(* CoDeSys 2.3 library: TcBACnetRev12.lib *)
(* Libraries: standard.lib 5.6.98 11:03:02, TcBase.lib 14.5.09 11:14:08, TcSystem.lib 21.1.15 09:22:54, TcUtilities.lib 6.1.15 15:45:04, TcTestAndSet.lib 23.2.09 11:50:08 *)

(* Global variable list: BACnet_Globals *)
VAR_GLOBAL
(* ADS read/write buffer for dynamic sized properties *)
	stBACnet_AdsBuffer		: ST_BACnet_GlobalAdsBuffer; (* 8kByte common ADS buffer used by function blocks that access BACnet over ADS *)
(* global linkable BACnet adapter *)
	fbBACnet_Adapter		: FB_BACnet_Adapter;
(* global visible BACnet adapter reference *)
	pBACnet_Adapter			: POINTER TO FB_BACnet_Adapter;
END_VAR
VAR_GLOBAL CONSTANT
(*********************************************
	Data field maximum
**********************************************)
	BACnet_MaxDayEntry			: UINT := 19;
	BACnet_MaxExSchEntries		: UINT := 9;
	BACnet_MaxTimeValues		: UINT := 9;
	BACnet_MaxObjIdList			: UINT := 1999;
	BACnet_MaxLogBufferEntries	: UINT := 499;
	BACnet_MaxDestinationArray	: UINT := 19;

(*********************************************
	error codes
**********************************************)
	BACnet_ERR_NO_ERROR				: UINT := 0;
	BACnet_ERR_NO_VALID_NET_ID		: UINT := 1;
	BACnet_ERR_WRONG_MAPPING		: UINT := 2;
	BACnet_ERR_OPERATIONAL			: UINT := 3;
	BACnet_ERR_NO_ETH_LINK			: UINT := 4;
	BACnet_ERR_NO_GATEWAY			: UINT := 5;
	BACnet_ERR_WOC_TRIGGER_UNSUP	: UINT := 6;
	BACnet_ERR_WOC_DISABLED			: UINT := 7;
	BACnet_ERR_INVALID_OBJECTID		: UINT := 8;
	BACnet_ERR_INVALID_OBJECTTYPE	: UINT := 10;
	BACnet_ERR_INVALID_CYCLETIME	: UINT := 11;
	BACnet_ERR_INVALID_PARAMETER	: UINT := 12;

(* errors with reset 20.. *)
	BACnet_ERR_PERSISTENT_WRITE		: UINT := 20;
	BACnet_ERR_INVALID_ADS_CONN		: UINT := 21;
	BACnet_ERR_CLIENT_TIMEOUT		: UINT := 22;
	BACnet_ERR_CLIENT_SERVICE		: UINT := 23;
	BACnet_ERR_WOC_TRIGGER_ACTIVE	: UINT := 24;
	BACnet_ERR_REVISION_READ		: UINT := 25;
	BACnet_ERR_PERSISTENT_PLC_WRITE	: UINT := 26;

(* ADS connection errors 30.. *)
	BACnet_ERR_ADS_NO_VALID_NET_ID	: UINT := 30; (* missing a valid Net ID *)
	BACnet_ERR_ADS_Data				: UINT := 31; (* ADS data length is wrong *)
	BACnet_ERR_ADS_Read				: UINT := 32; (* ADS read function was aborted *)
	BACnet_ERR_ADS_Write			: UINT := 33; (* ADS write function was aborted *)
	BACnet_ERR_ADS_ObjType			: UINT := 34; (* object type is wrong *)
	BACnet_ERR_ADS_ObjListEmpty		: UINT := 35; (* object list is empty *)
	BACnet_ERR_ADS_DeviceOP			: UINT := 36; (* device is not operational *)
	BACnet_ERR_ADS_NoDevice			: UINT := 37; (* no device object in object info list *)
	BACnet_ERR_ADS_ObjInstance		: UINT := 38; (* object list info is wrong *)
	BACnet_ERR_ADS_AmsPort			: UINT := 39; (* read AMS port is invalid (<1000) *)
	BACnet_ERR_ADS_ObjectId			: UINT := 40; (* object list info is wrong *)
	BACnet_ERR_ADS_LegacyStack		: UINT := 41; (* revision 6 stack detected (service is available from/above revision 9) *)
	BACnet_ERR_ADS_ObjIdMissmatch	: UINT := 42; (* object ID mapped and object list info are different *)
	BACnet_ERR_ADS_BufferSize		: UINT := 43; (* Property data larger than ADS buffer *)
	BACnet_ERR_ADS_SchedData		: UINT := 44; (* Wrong schedule property data *)
	BACnet_ERR_UnknownEventChoice	: UINT := 45; (* Unknown event choice type *)
	BACnet_ERR_UnknownEntryChoice	: UINT := 46; (* Unknown entry choice type *)
	BACnet_ERR_ADS_TooManyObjects	: UINT := 47; (* List of objects are longer than output list size *)
	BACnet_ERR_ADS_WrongEntrySize	: UINT := 48; (* expected entry size dosn't match read size *)
	BACnet_ERR_ADS_RecipientData	: UINT := 49; (* Invalid recipient data, device type expected *)
	BACnet_ERR_ADS_TooManyEntries	: UINT := 50; (* More entries than expected *)
	BACnet_ERR_ADS_NotEnoughEntries	: UINT := 51; (* Property incomplete, missing entries *)
	BACnet_ERR_ADS_Encoding			: UINT := 52; (* String encoding not supported *)
	BACnet_ERR_ADS_NoServerClient	: UINT := 53; (* Given ADS connection is not an server or client connection (expected bClient or bServer) *)
	BACnet_ERR_ADS_NoNotificationSink: UINT := 54; (* Given ADS connection is not an notification sink connection (expected bNSink) *)

(*********************************************
	other definitions
**********************************************)
	BACnet_ADSTimeOut			: TIME := t#15s;
	BACnet_PlcPersisTimeOut		: TIME := t#2m;
	BACnet_STRING_MAXLENGTH     : INT := 256;
	BACnet_ADSBufferSize		: INT := 8191; (* default 8kByte buffer *)

(* ADS index and groups *)
	BACnet_ADSIGRP_GET_OBJECT_LIST						: UDINT := 16#82400000;
	BACnet_ADSIGRP_CLIENT_COM_PARAMETER					: UDINT := 16#84000000;
	BACnet_ADSIGRP_DEV_R_GETADSPORTBYDEVID				: UDINT := 16#80000047; (* Get AMS Port BY Device ID *)
	BACnet_ADSIGRP_NTFSINK_EVENTNTF_CNT					: UDINT := 16#00000001;
	BACnet_ADSIGRP_NTFSINK_COVNTF_CNT					: UDINT := 16#00000002;
	BACnet_ADSIGRP_NTFSINK_EVENTNTF_READ				: UDINT := 16#00000003;
	BACnet_ADSIGRP_NTFSINK_COVNTF_READ					: UDINT := 16#00000004;
	BACnet_ADSIGRP_NTFSINK_EVENTNTF_DELETE				: UDINT := 16#00000005;
	BACnet_ADSIGRP_NTFSINK_COVNTF_DELETE				: UDINT := 16#00000006;
	BACnet_ADSIGRP_NTFSINK_EVENTNTF_INFO				: UDINT := 16#00000007;
	BACnet_ADSIGRP_NTFSINK_COVNTF_INFO					: UDINT := 16#00000008;
	BACnet_ADSIGRP_WRITE_NTFSINK_EVENTNTF_ACK			: UDINT := 16#00000009;
	BACnet_ADSIGRP_NTFSINK_W_EVENTNTF_ACK_BY_SEQUENCE	: UDINT := 16#0000000A;
	BACnet_ADSIGRP_NTFSINK_W_EVENTNTF_ACK_BY_PARAMETER	: UDINT := 16#0000000B;
	BACnet_ADSIGRP_NTFSINK_R_EVENTNTF_READ_BY_SEQUENCE	: UDINT := 16#0000000C;
	BACnet_ADSIGRP_NTFSINK_R_COVNTF_READ_BY_SEQUENCE	: UDINT := 16#0000000D;
	BACnet_ADSIGRP_NTFSINK_R_EVENTNTF_DELETE_BY_SEQUENCE: UDINT := 16#0000000E;
	BACnet_ADSIGRP_NTFSINK_R_COVNTF_DELETE_BY_SEQUENCE	: UDINT := 16#0000000F;


(* Object specifications *)
	arrBACnet_ObjectTypeNameShort : ARRAY[0..BACnetObjectType_ZCount] OF STRING(5) :=
		'AI' (* BACnetObjectType_AnalogInput :=0 *),
		'AO' (* BACnetObjectType_AnalogOutput :=1 *),
		'AV' (* BACnetObjectType_AnalogValue :=2 *),
		'BI' (* BACnetObjectType_BinaryInput :=3 *),
		'BO' (* BACnetObjectType_BinaryOutput :=4 *),
		'BV' (* BACnetObjectType_BinaryValue :=5 *),
		'CAL' (* BACnetObjectType_Calendar :=6 *),
		'CMD' (* BACnetObjectType_Command :=7 *),
		'DEV' (* BACnetObjectType_Device :=8 *),
		'EE' (* BACnetObjectType_EventEnrollment :=9 *),
		'FILE' (* BACnetObjectType_File :=10 *),
		'GROUP' (* BACnetObjectType_Group :=11 *),
		'LOOP' (* BACnetObjectType_Loop :=12 *),
		'MI' (* BACnetObjectType_MultiStateInput :=13 *),
		'MO' (* BACnetObjectType_MultiStateOutput :=14 *),
		'NC' (* BACnetObjectType_NotificationClass :=15 *),
		'PROG' (* BACnetObjectType_Program :=16 *),
		'SCHED' (* BACnetObjectType_Schedule :=17 *),
		'AVG' (* BACnetObjectType_Averaging :=18 *),
		'MV' (* BACnetObjectType_MultiStateValue :=19 *),
		'TLOG' (* BACnetObjectType_TrendLog :=20 *),
		'LP' (* BACnetObjectType_LifeSafetyPoint :=21 *),
		'LZ' (* BACnetObjectType_LifeSafetyZone :=22 *),
		'ACC' (* BACnetObjectType_Accumulator :=23 *),
		'PC' (* BACnetObjectType_PulseConverter :=24 *),
		'' (* BACnetObjectType_ZCount :=25 *);



END_VAR

(* Data type *)
TYPE E_BACNETACTION:
(
	BACnetAction_direct :=0,
	BACnetAction_reverse :=1
);
END_TYPE

(* Data type *)
TYPE E_BACNETADAPTERSTATUS :
(
	BACnetAdapterStatus_Init			:= 16#0,
	BACnetAdapterStatus_CheckIpAddr		:= 16#1,
	BACnetAdapterStatus_CheckParam		:= 16#2,
	BACnetAdapterStatus_GetGatewayMAC	:= 16#3,
	BACnetAdapterStatus_WaitGatewayMAC	:= 16#4,
	BACnetAdapterStatus_Complete		:= 16#8
);
END_TYPE

(* Data type *)
TYPE E_BACNETBINARYPV:
(
	BACnetBinaryPV_inactive :=0,
	BACnetBinaryPV_active :=1,
	BACnetBinaryPV_NULL := 2,
	BACnetBinaryPV_Nothing := 16#FFFF
);
END_TYPE

(* Data type *)
TYPE E_BACnetCalendarEntryChoice :
(
(*
	BACnetDate              DATE;
	BACnetDateRange   		dateRange;
	BACnetWeekNDay          weekNDay;
*)
	BACnetCalendarEntryChoice_date,
	BACnetCalendarEntryChoice_dateRange,
	BACnetCalendarEntryChoice_weekNDay
);
END_TYPE

(* Data type *)
TYPE E_BACnetCalendarEntryType : (* Not a BACnet-Stack type! *)
(
	BACnetCalendarEntryType_None,
	BACnetCalendarEntryType_Ref,
	BACnetCalendarEntryType_Date,
	BACnetCalendarEntryType_DateRange,
	BACnetCalendarEntryType_WeekNDay
);
END_TYPE

(* Data type *)
TYPE E_BACNETDATATYPES:
(
	BACnetDataType_Null :=0,
	BACnetDataType_Bool :=1,
	BACnetDataType_UnsignedInteger :=2,
	BACnetDataType_SignedInteger :=3,
	BACnetDataType_Real :=4,
	BACnetDataType_Double :=5,
	BACnetDataType_OctetString :=6,
	BACnetDataType_CharacterStringExt :=7,
	BACnetDataType_BitString :=8,
	BACnetDataType_Enumerated :=9,
	BACnetDataType_Date :=10,
	BACnetDataType_Time :=11,
	BACnetDataType_ObjectIdentifier :=12,
	BACnetDataType_DateTime :=14,
	BACnetDataType_ArrayIndex :=15,
	BACnetDataType_CalendarEntry :=16,
	BACnetDataType_ObjectType :=17,
	BACnetDataType_EventTransitionBits :=18,
	BACnetDataType_ActionList :=19,
	BACnetDataType_StatusFlags :=20,
	BACnetDataType_EventState :=21,
	BACnetDataType_Reliability :=22,
	BACnetDataType_Polarity :=23,
	BACnetDataType_EngineeringUnits :=25,
	BACnetDataType_PriorityValue :=26,
	BACnetDataType_LimitEnable :=27,
	BACnetDataType_NotifyType :=29,
	BACnetDataType_TimeStamp :=30,
	BACnetDataType_DeviceObjectPropertyReference :=31,
	BACnetDataType_DeviceStatus :=32,
	BACnetDataType_ServicesSupported :=33,
	BACnetDataType_ObjectTypesSupported :=34,
	BACnetDataType_Segmentation :=35,
	BACnetDataType_VTClass :=36,
	BACnetDataType_VTSession :=37,
	BACnetDataType_SessionKey :=38,
	BACnetDataType_Recipient :=39,
	BACnetDataType_AddressBinding :=40,
	BACnetDataType_COVSubscription :=41,
	BACnetDataType_EventType :=42,
	BACnetDataType_EventParameter :=43,
	BACnetDataType_FileAccessMethod :=44,
	BACnetDataType_ReadAccessSpecification :=45,
	BACnetDataType_ReadAccessResult :=46,
	BACnetDataType_ObjectPropertyReference :=47,
	BACnetDataType_SetpointReference :=48,
	BACnetDataType_Destination :=49,
	BACnetDataType_ProgramState :=50,
	BACnetDataType_ProgramRequest :=51,
	BACnetDataType_ProgramError :=52,
	BACnetDataType_DateRange :=53,
	BACnetDataType_DailySchedule :=54,
	BACnetDataType_SpecialEvent :=55,
	BACnetDataType_ClientCOV :=56,
	BACnetDataType_LogRecord :=57,
	BACnetDataType_LifeSafetyState :=58,
	BACnetDataType_LifeSafetyMode :=59,
	BACnetDataType_SilencedState :=60,
	BACnetDataType_LifeSafetyOperation :=61,
	BACnetDataType_BinaryPV :=62,
	BACnetDataType_DaysOfWeek :=63,
	BACnetDataType_WeekNDay :=64,
	BACnetDataType_TimeValue :=65,
	BACnetDataType_Value :=66,
	BACnetDataType_Address :=67,
	BACnetDataType_PropertyIdentifier :=68,
	BACnetDataType_EnumerationValueType :=69,
	BACnetDataType_BitFieldBit :=70,
	BACnetDataType_LogDatum :=71,
	BACnetDataType_AnyType :=72,
	BACnetDataType_PresentValue :=73,
	BACnetDataType_ContextTag :=74,
	BACnetDataType_ValueChoice :=75,
	BACnetDataType_LogStatus :=76,
	BACnetDataType_RecipientProcess :=77,
	BACnetDataType_SubscribeCOVPropertyRequest :=78,
	BACnetDataType_PropertyReference :=79,
	BACnetDataType_PropertyResult :=80,
	BACnetDataType_DeviceObjectPropertyValue :=81,
	BACnetDataType_COVNotificationRequest :=82,
	BACnetDataType_EventNotificationRequest :=83,
	BACnetDataType_NotificationParameters :=84,
	BACnetDataType_Change_of_Bitstring :=85,
	BACnetDataType_Change_of_State :=86,
	BACnetDataType_Change_of_Value :=87,
	BACnetDataType_Command_failure :=88,
	BACnetDataType_Floating_limit :=89,
	BACnetDataType_Out_of_Range :=90,
	BACnetDataType_PropertyValue :=91,
	BACnetDataType_Complex_Tag :=92,
	BACnetDataType_Change_of_life_safety :=93,
	BACnetDataType_Extended :=94,
	BACnetDataType_Buffer_ready :=95,
	BACnetDataType_Unsigned_range :=96,
	BACnetDataType_PropertyResultValue :=97,
	BACnetDataType_ServiceCOVPropSubscription :=98,
	BACnetDataType_ServiceCOVSubscription :=99,
	BACnetDataType_COVNotification :=100,
	BACnetDataType_AcknowledgeAlarmRequest :=101,
	BACnetDataType_VTOpenRequest :=102,
	BACnetDataType_Prescale :=103,
	BACnetDataType_Scale :=104,
	BACnetDataType_Action :=105,
	BACnetDataType_Error :=106,
	BACnetDataType_ErrorType :=107,
	BACnetDataType_ErrorClass :=108,
	BACnetDataType_ErrorCode :=109,
	BACnetDataType_RejectReason :=110,
	BACnetDataType_AbortReason :=111,
	BACnetDataType_BDTEntry :=112,
	BACnetDataType_IpEntry :=113,
	BACnetDataType_MaskEntry :=114,
	BACnetDataType_EthernetAddress := 115,
	BACnetDataType_LonTalkAddress := 116,
	BACnetDataType_LonTalkNeuronId := 117,
	BACnetDataType_NodeType := 118,
	BACnetDataType_DeviceObjectReference := 119,
	BACnetDataType_ActionCommand := 120,
	BACnetDataType_GetEventInformation := 121,
	BACnetDataType_GetEnrollmentSummaryCriteria := 122,
	BACnetDataType_GetEnrollmentSummaryCriteriaResponse := 123,
	BACnetDataType_DeviceCommunicationControl := 124,
	BACnetDataType_Int16 := 125,
	BACnetDataType_UInt16 := 126,
	BACnetDataType_UInt8 := 127,
	BACnetDataType_TypeInt8 := 128,
	BACnetDataType_Byte := 129,
	BACnetDataType_FDTEntry := 130,
	BACnetDataType_Address_3 := 131,
	BACnetDataType_Address_4 := 132,
	BACnetDataType_Address_5 := 133,
	BACnetDataType_PersistentDataState := 134,
	BACnetDataType_FallbackRealValue := 135,
	BACnetDataType_FallbackBinaryValue := 136,
	BACnetDataType_RealNull := 137, (* PresentValue in AnalogObj *)
	BACnetDataType_EnumeratedNull := 138, (* PresentValue in BinaryObj *)
	BACnetDataType_UnsignedIntegerNull := 139, (* PresentValue in Multistate *)
	BACnetDataType_Unknown := 140,
	BACnetDataType_DiagnosisPerformance := 200,
	BACnetDataType_DiagnosisEthStatistics := 201,
	BACnetDataType_FrameStatistics := 202,
	BACnetDataType_Info := 203,
	BACnetDataType_Diagnosis := 204,
	BACnetDataType_TcIoEthStatistic := 205,
	BACnetDataType_TcIoEthTxRxErrorCount := 206,
	BACnetDataType_TcIoEthPortStatistic := 207,
	BACnetDataType_ServerStatistics := 208,
	BACnetDataType_FrameServicesDiag := 209,
	BACnetDataType_UnsignedIntegerArr :=258,
	BACnetDataType_CharacterStringExtArr :=263,
	BACnetDataType_ObjectIdentifierArr :=268,
	BACnetDataType_CalendarEntryArr :=272,
	BACnetDataType_ActionListArr :=275,
	BACnetDataType_PriorityValueArr :=282,
	BACnetDataType_TimeStampArr :=286,
	BACnetDataType_DeviceObjectPropertyReferenceArr :=287,
	BACnetDataType_VTClassArr :=292,
	BACnetDataType_VTSessionArr :=293,
	BACnetDataType_SessionKeyArr :=294,
	BACnetDataType_RecipientArr :=295,
	BACnetDataType_AddressBindingArr :=296,
	BACnetDataType_COVSubscriptionArr :=297,
	BACnetDataType_ReadAccessSpecificationArr :=301,
	BACnetDataType_ReadAccessResultArr :=302,
	BACnetDataType_DestinationArr :=305,
	BACnetDataType_SpecialEventArr :=311,
	BACnetDataType_LogRecordArr :=313,
	BACnetDataType_LifeSafetyStateArr :=314,
	BACnetDataType_TimeValueArr :=321,
	BACnetDataType_UnsignedIntegerList :=514,
	BACnetDataType_CharacterStringExtList :=519,
	BACnetDataType_ReadAccessSpecificationList :=557,
	BACnetDataType_ReadAccessResultList :=558,
	BACnetDataType_SpecialEventList :=567,
	BACnetDataType_LogRecordList :=569,
	BACnetDataType_TimeValueList :=577,
	BACnetDataType_ValueList :=578,
	BACnetDataType_LogDatumList :=583,
	BACnetDataType_PropertyReferenceList :=591,
	BACnetDataType_PropertyResultList :=592,
	BACnetDataType_COVNotificationRequestList :=594,
	BACnetDataType_EventNotificationRequestList :=595,
	BACnetDataType_PropertyValueList :=603,
	BACnetDataType_DailyScheduleList :=1089
);
END_TYPE

(* Data type *)
TYPE E_BACNETDAYSOFWEEKBITS :
(
	BACnetDaysOfWeekBits_Monday		:= 0,
	BACnetDaysOfWeekBits_Tuesday	:= 1,
	BACnetDaysOfWeekBits_Wednesday	:= 2,
	BACnetDaysOfWeekBits_Thursday	:= 3,
	BACnetDaysOfWeekBits_Friday		:= 4,
	BACnetDaysOfWeekBits_Saturday	:= 5,
	BACnetDaysOfWeekBits_Sunday		:= 6
);
END_TYPE

(* Data type *)
TYPE E_BACNETDEVICESTATUS:
(
	BACnetDeviceStatus_Operational :=0,
	BACnetDeviceStatus_OperationalReadOnly :=1,
	BACnetDeviceStatus_DownloadRequired :=2,
	BACnetDeviceStatus_DownloadInProgress :=3,
	BACnetDeviceStatus_NonOperational :=4,
	BACnetDeviceStatus_BackupInProgress :=5
);
END_TYPE

(* Data type *)
TYPE E_BACNETEVENTSTATE:
(
	BACnetEventState_state_normal :=0,
	BACnetEventState_fault :=1,
	BACnetEventState_offnormal :=2,
	BACnetEventState_high_limit :=3,
	BACnetEventState_low_limit :=4,
	BACnetEventState_life_safety_alarm :=5
);
END_TYPE

(* Data type *)
TYPE E_BACNETEVENTTRANSITIONBIT:
(
	BACnetEventTransitionBit_to_offnormal :=0,
	BACnetEventTransitionBit_to_fault :=1,
	BACnetEventTransitionBit_to_normal :=2
);
END_TYPE

(* Data type *)
TYPE E_BACNETEVENTTYPE:
(
	BACnetEventType_change_of_bitstring :=0,
	BACnetEventType_change_of_state :=1,
	BACnetEventType_change_of_value :=2,
	BACnetEventType_command_failure :=3,
	BACnetEventType_floating_limit :=4,
	BACnetEventType_out_of_range :=5,
	BACnetEventType_complex_event_type :=6,
	BACnetEventType_deprecated7 :=7,
	BACnetEventType_change_of_life_safety :=8,
	BACnetEventType_enumeration :=9,
	BACnetEventType_buffer_ready :=10,
	BACnetEventType_unsigned_range :=11,
	BACnetEventType_reserved12 := 12,
	BACnetEventType_access_event := 13,
	BACnetEventType_double_out_of_range := 14,
	BACnetEventType_signed_out_of_range := 15,
	BACnetEventType_unsigned_out_of_range := 16,
	BACnetEventType_change_of_characterstring := 17,
	BACnetEventType_change_of_state_flags := 18
);
END_TYPE

(* Data type *)
TYPE E_BACNETFILEACCESSMETHOD:
(
	BACnetFileAccessMethod_record_access :=0,
	BACnetFileAccessMethod_stream_access :=1
);
END_TYPE

(* Data type *)
TYPE E_BACNETLIFESAFETYMODE:
(
	BACnetLifeSafetyMode_off :=0,
	BACnetLifeSafetyMode_on :=1,
	BACnetLifeSafetyMode_test :=2,
	BACnetLifeSafetyMode_manned :=3,
	BACnetLifeSafetyMode_unmanned :=4,
	BACnetLifeSafetyMode_armed :=5,
	BACnetLifeSafetyMode_disarmed :=6,
	BACnetLifeSafetyMode_prearmed :=7,
	BACnetLifeSafetyMode_slow :=8,
	BACnetLifeSafetyMode_fast :=9,
	BACnetLifeSafetyMode_disconnected :=10,
	BACnetLifeSafetyMode_enabled :=11,
	BACnetLifeSafetyMode_disabled :=12,
	BACnetLifeSafetyMode_automatic_release_disabled :=13,
	BACnetLifeSafetyMode_mode_default :=14
);
END_TYPE

(* Data type *)
TYPE E_BACNETLIFESAFETYOPERATION:
(
	BACnetLifeSafetyOperation_none :=0,
	BACnetLifeSafetyOperation_silence :=1,
	BACnetLifeSafetyOperation_silence_audible :=2,
	BACnetLifeSafetyOperation_silence_visual :=3,
	BACnetLifeSafetyOperation_reset :=4,
	BACnetLifeSafetyOperation_reset_alarm :=5,
	BACnetLifeSafetyOperation_reset_fault :=6,
	BACnetLifeSafetyOperation_unsilence := 7,
	BACnetLifeSafetyOperation_unsilence_audible := 8,
	BACnetLifeSafetyOperation_unsilence_visual := 9
);
END_TYPE

(* Data type *)
TYPE E_BACNETLIMITENABLEBITS:
(
	BACnetLimitEnableBits_lowLimit :=0,
	BACnetLimitEnableBits_highLimit :=1
);
END_TYPE

(* Data type *)
TYPE E_BACNETLOGGINGTYPE :
(
	BACnetLoggingType_cov,
	BACnetLoggingType_polled,
	BACnetLoggingType_triggered
);
END_TYPE

(* Data type *)
TYPE E_BACnetLogRecordChoice :
(
(*
enum BACnetLogRecordChoice
{
      logStatus,              // [0] BACnetLogStatus,
      booleanValue,           // [1] BOOL,
      realValue,              // [2] REAL,
      enumValue,              // [3] ENUMERATED, __ Optionally limited to 32 bits
      unsignedValue,          // [4] Unsigned, __ Optionally limited to 32 bits
      signedValue,            // [5] INTEGER, __ Optionally limited to 32 bits
      bitstringValue,         // [6] BIT STRING, __ Optionally limited to 32 bits
      nullValue,              // [7] NULL,
      failure,                // [8] Error,
      timeChange,             // [9] REAL,
      anyValue,               // [10] ABSTRACT_SYNTAX.&Type __ Optional
};
*)
	BACnetLogRecordChoice_logStatus 	:= 0, (* BACnetLogStatus *)
	BACnetLogRecordChoice_booleanValue := 1, (*  BOOL, *)
	BACnetLogRecordChoice_realValue	:= 2, (*  REAL, *)
	BACnetLogRecordChoice_enumValue	:= 3, (*  ENUMERATED, __ Optionally limited TO 32 bits *)
	BACnetLogRecordChoice_unsignedValue:= 4, (*  Unsigned, __ Optionally limited TO 32 bits *)
	BACnetLogRecordChoice_signedValue	:= 5, (*  INTEGER, __ Optionally limited TO 32 bits *)
	BACnetLogRecordChoice_bitstringValue:= 6, (*  BIT STRING, __ Optionally limited TO 32 bits *)
	BACnetLogRecordChoice_nullValue	:= 7, (*  NULL, *)
	BACnetLogRecordChoice_failure		:= 8, (*  Error, *)
	BACnetLogRecordChoice_timeChange	:= 9, (*  REAL, *)
	BACnetLogRecordChoice_anyValue		:= 10 (*  ABSTRACT_SYNTAX.&TYPE __ Optional *)
);
END_TYPE

(* Data type *)
TYPE E_BACNETLOOPMODE :
(
	BACnetLoopMode_None,		(* LOOP object has unknown parameter settings *)
	BACnetLoopMode_Ideal,		(* Controller is in ideal form: P, I and D are in parallel junktion; unit of P, I and D is [1] (Kp, Ki, Kd) *)
	BACnetLoopMode_Standard		(* Controller works in standard form (most industrial applications): P parameter is applied to I and D; unit of I and D is time based [s] (Kp, Ti, Td) *)
);
END_TYPE

(* Data type *)
TYPE E_BACNETNOTIFYTYPE:
(
	BACnetNotifyType_alarm :=0,
	BACnetNotifyType_notify_event :=1,
	BACnetNotifyType_ack_notification :=2
);
END_TYPE

(* Data type *)
TYPE E_BACNETOBJECTSUPPORTEDBITS:
(
	BACnetObjectSupportedBits_AnalogInput :=0,
	BACnetObjectSupportedBits_AnalogOutput :=1,
	BACnetObjectSupportedBits_AnalogValue :=2,
	BACnetObjectSupportedBits_BinaryInput :=3,
	BACnetObjectSupportedBits_BinaryOutput :=4,
	BACnetObjectSupportedBits_BinaryValue :=5,
	BACnetObjectSupportedBits_Calendar :=6,
	BACnetObjectSupportedBits_Command :=7,
	BACnetObjectSupportedBits_Device :=8,
	BACnetObjectSupportedBits_EventEnrollment :=9,
	BACnetObjectSupportedBits_File :=10,
	BACnetObjectSupportedBits_Group :=11,
	BACnetObjectSupportedBits_Loop :=12,
	BACnetObjectSupportedBits_MultiStateInput :=13,
	BACnetObjectSupportedBits_MultiStateOutput :=14,
	BACnetObjectSupportedBits_NotificationClass :=15,
	BACnetObjectSupportedBits_Program :=16,
	BACnetObjectSupportedBits_Schedule :=17,
	BACnetObjectSupportedBits_Averaging :=18,
	BACnetObjectSupportedBits_MultiStateValue :=19,
	BACnetObjectSupportedBits_TrendLog :=20,
	BACnetObjectSupportedBits_LifeSafetyPoint :=21,
	BACnetObjectSupportedBits_LifeSafetyZone :=22,
	BACnetObjectSupportedBits_Accumulator := 23,
	BACnetObjectSupportedBits_PulseConverter := 24,
	BACnetObjectSupportedBits_EventLog := 25,
	BACnetObjectSupportedBits_GlobalGroup := 26,
	BACnetObjectSupportedBits_TrendLogMultiple := 27,
	BACnetObjectSupportedBits_LoadControl := 28,
	BACnetObjectSupportedBits_StructuredView := 29,
	BACnetObjectSupportedBits_AccessDoor := 30,
	BACnetObjectSupportedBits_unassigend31 := 31,
	BACnetObjectSupportedBits_AccessCredential := 32,
	BACnetObjectSupportedBits_AccessPoint := 33,
	BACnetObjectSupportedBits_AccessRights := 34,
	BACnetObjectSupportedBits_AccessUser := 35,
	BACnetObjectSupportedBits_AccessZone := 36,
	BACnetObjectSupportedBits_CredentialDataInput := 37,
	BACnetObjectSupportedBits_NetworkSecurity := 38,
	BACnetObjectSupportedBits_BitStringValue := 39,
	BACnetObjectSupportedBits_CharacterStringValue := 40,
	BACnetObjectSupportedBits_DatePatternValue := 41,
	BACnetObjectSupportedBits_DateValue := 42,
	BACnetObjectSupportedBits_DateTimePatternValue := 43,
	BACnetObjectSupportedBits_DateTimeValue := 44,
	BACnetObjectSupportedBits_IntegerValue := 45,
	BACnetObjectSupportedBits_LargeAnalogValue := 46,
	BACnetObjectSupportedBits_OctetStringValue := 47,
	BACnetObjectSupportedBits_PositiveIntegerValue := 48,
	BACnetObjectSupportedBits_TimePatternValue := 49,
	BACnetObjectSupportedBits_TimeValue := 50,
	BACnetObjectSupportedBits_NetworkPort := 51,
	BACnetObjectSupportedBits_AlertEnrollment := 52,
	BACnetObjectSupportedBits_Channel := 53
);
END_TYPE

(* Data type *)
TYPE E_BACNETOBJECTTYPE:
(
	BACnetObjectType_AnalogInput :=0,
	BACnetObjectType_AnalogOutput :=1,
	BACnetObjectType_AnalogValue :=2,
	BACnetObjectType_BinaryInput :=3,
	BACnetObjectType_BinaryOutput :=4,
	BACnetObjectType_BinaryValue :=5,
	BACnetObjectType_Calendar :=6,
	BACnetObjectType_Command :=7,
	BACnetObjectType_Device :=8,
	BACnetObjectType_EventEnrollment :=9,
	BACnetObjectType_File :=10,
	BACnetObjectType_Group :=11,
	BACnetObjectType_Loop :=12,
	BACnetObjectType_MultiStateInput :=13,
	BACnetObjectType_MultiStateOutput :=14,
	BACnetObjectType_NotificationClass :=15,
	BACnetObjectType_Program :=16,
	BACnetObjectType_Schedule :=17,
	BACnetObjectType_Averaging :=18,
	BACnetObjectType_MultiStateValue :=19,
	BACnetObjectType_TrendLog :=20,
	BACnetObjectType_LifeSafetyPoint :=21,
	BACnetObjectType_LifeSafetyZone :=22,
	BACnetObjectType_Accumulator :=23,
	BACnetObjectType_PulseConverter :=24,
	BACnetObjectType_EventLog := 25,
	BACnetObjectType_GlobalGroup := 26,
	BACnetObjectType_TrendLogMultiple := 27,
	BACnetObjectType_LoadControl := 28,
	BACnetObjectType_StructuredView := 29,
	BACnetObjectType_AccessDoor := 30,
	BACnetObjectType_unassigend31 := 31,
	BACnetObjectType_AccessCredential := 32,
	BACnetObjectType_AccessPoint := 33,
	BACnetObjectType_AccessRights := 34,
	BACnetObjectType_AccessUser := 35,
	BACnetObjectType_AccessZone := 36,
	BACnetObjectType_CredentialDataInput := 37,
	BACnetObjectType_NetworkSecurity := 38,
	BACnetObjectType_BitStringValue := 39,
	BACnetObjectType_CharacterStringValue := 40,
	BACnetObjectType_DatePatternValue := 41,
	BACnetObjectType_DateValue := 42,
	BACnetObjectType_DateTimePatternValue := 43,
	BACnetObjectType_DateTimeValue := 44,
	BACnetObjectType_IntegerValue := 45,
	BACnetObjectType_LargeAnalogValue := 46,
	BACnetObjectType_OctetStringValue := 47,
	BACnetObjectType_PositiveIntegerValue := 48,
	BACnetObjectType_TimePatternValue := 49,
	BACnetObjectType_TimeValue := 50,
	BACnetObjectType_NetworkPort := 51,
	BACnetObjectType_AlertEnrollment := 52,
	BACnetObjectType_Channel := 53,


	(* keep at the end of list! *)
	BACnetObjectType_ZCount
);
END_TYPE

(* Data type *)
TYPE E_BACNETPERSISTENTDATASTATE :
(
	BACnetPersistentData_Disabled,
	BACnetPersistentData_Initialize,
	BACnetPersistentData_NoChange,
	BACnetPersistentData_Ready,
	BACnetPersistentData_Write,
	BACnetPersistentData_Writing
);
END_TYPE

(* Data type *)
TYPE E_BACNETPIDTUNINGMODE :
(
	BACnetPIDTuningMode_P,
	BACnetPIDTuningMode_PI,
	BACnetPIDTuningMode_PD,
	BACnetPIDTuningMode_PID
);
END_TYPE

(* Data type *)
TYPE E_BACNETPOLARITY:
(
	BACnetPolarity_normal :=0,
	BACnetPolarity_reverse :=1
);
END_TYPE

(* Data type *)
TYPE E_BACNETPRIORITY:
(
	BACnetPriority_None :=0,
	BACnetPriority_1 :=1,
	BACnetPriority_2 :=2,
	BACnetPriority_3 :=3,
	BACnetPriority_4 :=4,
	BACnetPriority_5 :=5,
	BACnetPriority_6 :=6,
	BACnetPriority_7 :=7,
	BACnetPriority_8 :=8,
	BACnetPriority_9 :=9,
	BACnetPriority_10 :=10,
	BACnetPriority_11 :=11,
	BACnetPriority_12 :=12,
	BACnetPriority_13 :=13,
	BACnetPriority_14 :=14,
	BACnetPriority_15 :=15,
	BACnetPriority_16 :=16
);
END_TYPE

(* Data type *)
TYPE E_BACNETPROGRAMERROR:
(
	BACnetProgramError_program_normal :=0,
	BACnetProgramError_load_failed :=1,
	BACnetProgramError_progerror_internal :=2,
	BACnetProgramError_program :=3,
	BACnetProgramError_other :=4
);
END_TYPE

(* Data type *)
TYPE E_BACNETPROGRAMREQUEST:
(
	BACnetProgramRequest_ready :=0,
	BACnetProgramRequest_load :=1,
	BACnetProgramRequest_run :=2,
	BACnetProgramRequest_halt :=3,
	BACnetProgramRequest_restart :=4,
	BACnetProgramRequest_unload :=5
);
END_TYPE

(* Data type *)
TYPE E_BACNETPROGRAMSTATE:
(
	BACnetProgramState_idle :=0,
	BACnetProgramState_loading :=1,
	BACnetProgramState_running :=2,
	BACnetProgramState_waiting :=3,
	BACnetProgramState_halted :=4,
	BACnetProgramState_unloading :=5
);
END_TYPE

(* Data type *)
TYPE E_BACNETPROPERTYIDENTIFIER:
(
	BACnetPropertyIdentifier_AckedTransitions 	:=	0	,
	BACnetPropertyIdentifier_AckRequired 	:=	1	,
	BACnetPropertyIdentifier_Action 	:=	2	,
	BACnetPropertyIdentifier_ActionText 	:=	3	,
	BACnetPropertyIdentifier_ActiveText 	:=	4	,
	BACnetPropertyIdentifier_ActiveVTSessions 	:=	5	,
	BACnetPropertyIdentifier_AlarmValue 	:=	6	,
	BACnetPropertyIdentifier_AlarmValues 	:=	7	,
	BACnetPropertyIdentifier_All 	:=	8	,
	BACnetPropertyIdentifier_AllWritesSuccessful 	:=	9	,
	BACnetPropertyIdentifier_ApduSegmentTimeout 	:=	10	,
	BACnetPropertyIdentifier_ApduTimeout 	:=	11	,
	BACnetPropertyIdentifier_ApplicationSoftwareVersion 	:=	12	,
	BACnetPropertyIdentifier_Archive 	:=	13	,
	BACnetPropertyIdentifier_Bias 	:=	14	,
	BACnetPropertyIdentifier_ChangeOfStateCount 	:=	15	,
	BACnetPropertyIdentifier_ChangeOfStateTime 	:=	16	,
	BACnetPropertyIdentifier_NotificationClass 	:=	17	,
	BACnetPropertyIdentifier_Reserved18 	:=	18	,
	BACnetPropertyIdentifier_ControlledVariableReference 	:=	19	,
	BACnetPropertyIdentifier_ControlledVariableUnits 	:=	20	,
	BACnetPropertyIdentifier_ControlledVariableValue 	:=	21	,
	BACnetPropertyIdentifier_CovIncrement 	:=	22	,
	BACnetPropertyIdentifier_DateList 	:=	23	,
	BACnetPropertyIdentifier_DaylightSavingsStatus 	:=	24	,
	BACnetPropertyIdentifier_Deadband 	:=	25	,
	BACnetPropertyIdentifier_DerivativeConstant 	:=	26	,
	BACnetPropertyIdentifier_DerivativeConstantUnits 	:=	27	,
	BACnetPropertyIdentifier_Description 	:=	28	,
	BACnetPropertyIdentifier_DescriptionOfHalt 	:=	29	,
	BACnetPropertyIdentifier_DeviceAddressBinding 	:=	30	,
	BACnetPropertyIdentifier_DeviceType 	:=	31	,
	BACnetPropertyIdentifier_EffectivePeriod 	:=	32	,
	BACnetPropertyIdentifier_ElapsedActiveTime 	:=	33	,
	BACnetPropertyIdentifier_ErrorLimit 	:=	34	,
	BACnetPropertyIdentifier_EventEnable 	:=	35	,
	BACnetPropertyIdentifier_EventState 	:=	36	,
	BACnetPropertyIdentifier_EventType 	:=	37	,
	BACnetPropertyIdentifier_ExceptionSchedule 	:=	38	,
	BACnetPropertyIdentifier_FaultValues 	:=	39	,
	BACnetPropertyIdentifier_FeedbackValue 	:=	40	,
	BACnetPropertyIdentifier_FileAccessMethod 	:=	41	,
	BACnetPropertyIdentifier_FileSize 	:=	42	,
	BACnetPropertyIdentifier_FileType 	:=	43	,
	BACnetPropertyIdentifier_FirmwareRevision 	:=	44	,
	BACnetPropertyIdentifier_HighLimit 	:=	45	,
	BACnetPropertyIdentifier_InactiveText 	:=	46	,
	BACnetPropertyIdentifier_InProcess 	:=	47	,
	BACnetPropertyIdentifier_InstanceOf 	:=	48	,
	BACnetPropertyIdentifier_IntegralConstant 	:=	49	,
	BACnetPropertyIdentifier_IntegralConstantUnits 	:=	50	,
	BACnetPropertyIdentifier_IssueConfirmedNotifications 	:=	51	,
	BACnetPropertyIdentifier_LimitEnable 	:=	52	,
	BACnetPropertyIdentifier_ListOfGroupMembers 	:=	53	,
	BACnetPropertyIdentifier_ListOfObjectPropertyReferences 	:=	54	,
	BACnetPropertyIdentifier_ListOfSessionKeys 	:=	55	,
	BACnetPropertyIdentifier_LocalDate 	:=	56	,
	BACnetPropertyIdentifier_LocalTime 	:=	57	,
	BACnetPropertyIdentifier_Location 	:=	58	,
	BACnetPropertyIdentifier_LowLimit 	:=	59	,
	BACnetPropertyIdentifier_ManipulatedVariableReference 	:=	60	,
	BACnetPropertyIdentifier_MaximumOutput 	:=	61	,
	BACnetPropertyIdentifier_MaxApduLengthAccepted 	:=	62	,
	BACnetPropertyIdentifier_MaxInfoFrames 	:=	63	,
	BACnetPropertyIdentifier_MaxMaster 	:=	64	,
	BACnetPropertyIdentifier_MaxPresValue 	:=	65	,
	BACnetPropertyIdentifier_MinimumOffTime 	:=	66	,
	BACnetPropertyIdentifier_MinimumOnTime 	:=	67	,
	BACnetPropertyIdentifier_MinimumOutput 	:=	68	,
	BACnetPropertyIdentifier_MinPresValue 	:=	69	,
	BACnetPropertyIdentifier_ModelName 	:=	70	,
	BACnetPropertyIdentifier_ModificationDate 	:=	71	,
	BACnetPropertyIdentifier_NotifyType 	:=	72	,
	BACnetPropertyIdentifier_NumberOfAPDURetries 	:=	73	,
	BACnetPropertyIdentifier_NumberOfStates 	:=	74	,
	BACnetPropertyIdentifier_ObjectIdentifier 	:=	75	,
	BACnetPropertyIdentifier_ObjectList 	:=	76	,
	BACnetPropertyIdentifier_ObjectName 	:=	77	,
	BACnetPropertyIdentifier_ObjectPropertyReference 	:=	78	,
	BACnetPropertyIdentifier_ObjectType 	:=	79	,
	BACnetPropertyIdentifier_Optional 	:=	80	,
	BACnetPropertyIdentifier_OutOfService 	:=	81	,
	BACnetPropertyIdentifier_OutputUnits 	:=	82	,
	BACnetPropertyIdentifier_EventParameters 	:=	83	,
	BACnetPropertyIdentifier_Polarity 	:=	84	,
	BACnetPropertyIdentifier_PresentValue 	:=	85	,
	BACnetPropertyIdentifier_Priority 	:=	86	,
	BACnetPropertyIdentifier_PriorityArray 	:=	87	,
	BACnetPropertyIdentifier_PriorityForWriting 	:=	88	,
	BACnetPropertyIdentifier_ProcessIdentifier 	:=	89	,
	BACnetPropertyIdentifier_ProgramChange 	:=	90	,
	BACnetPropertyIdentifier_ProgramLocation 	:=	91	,
	BACnetPropertyIdentifier_ProgramState 	:=	92	,
	BACnetPropertyIdentifier_ProportionalConstant 	:=	93	,
	BACnetPropertyIdentifier_ProportionalConstantUnits 	:=	94	,
	BACnetPropertyIdentifier_ProtocolConformanceClass 	:=	95	,
	BACnetPropertyIdentifier_ProtocolObjectTypesSupported 	:=	96	,
	BACnetPropertyIdentifier_ProtocolServicesSupported 	:=	97	,
	BACnetPropertyIdentifier_ProtocolVersion 	:=	98	,
	BACnetPropertyIdentifier_ReadOnly 	:=	99	,
	BACnetPropertyIdentifier_ReasonForHalt 	:=	100	,
	BACnetPropertyIdentifier_Recipient 	:=	101	,
	BACnetPropertyIdentifier_RecipientList 	:=	102	,
	BACnetPropertyIdentifier_Reliability 	:=	103	,
	BACnetPropertyIdentifier_RelinquishDefault 	:=	104	,
	BACnetPropertyIdentifier_Required 	:=	105	,
	BACnetPropertyIdentifier_Resolution 	:=	106	,
	BACnetPropertyIdentifier_SegmentationSupported 	:=	107	,
	BACnetPropertyIdentifier_Setpoint 	:=	108	,
	BACnetPropertyIdentifier_SetpointReference 	:=	109	,
	BACnetPropertyIdentifier_StateText 	:=	110	,
	BACnetPropertyIdentifier_StatusFlags 	:=	111	,
	BACnetPropertyIdentifier_SystemStatus 	:=	112	,
	BACnetPropertyIdentifier_TimeDelay 	:=	113	,
	BACnetPropertyIdentifier_TimeOfActiveTimeReset 	:=	114	,
	BACnetPropertyIdentifier_TimeOfStateCountReset 	:=	115	,
	BACnetPropertyIdentifier_TimeSynchronizationRecipients 	:=	116	,
	BACnetPropertyIdentifier_Units 	:=	117	,
	BACnetPropertyIdentifier_UpdateInterval 	:=	118	,
	BACnetPropertyIdentifier_UtcOffset 	:=	119	,
	BACnetPropertyIdentifier_VendorIdentifier 	:=	120	,
	BACnetPropertyIdentifier_VendorName 	:=	121	,
	BACnetPropertyIdentifier_VtClassesSupported 	:=	122	,
	BACnetPropertyIdentifier_WeeklySchedule 	:=	123	,
	BACnetPropertyIdentifier_AttemptedSamples 	:=	124	,
	BACnetPropertyIdentifier_AverageValue 	:=	125	,
	BACnetPropertyIdentifier_BufferSize 	:=	126	,
	BACnetPropertyIdentifier_ClientCovIncrement 	:=	127	,
	BACnetPropertyIdentifier_CovResubscriptionInterval 	:=	128	,
	BACnetPropertyIdentifier_CurrentNotifyTime 	:=	129	,
	BACnetPropertyIdentifier_EventTimeStamps 	:=	130	,
	BACnetPropertyIdentifier_LogBuffer 	:=	131	,
	BACnetPropertyIdentifier_LogDeviceObjectProperty 	:=	132	,
	BACnetPropertyIdentifier_Enable 	:=	133	,
	BACnetPropertyIdentifier_LogInterval 	:=	134	,
	BACnetPropertyIdentifier_MaximumValue 	:=	135	,
	BACnetPropertyIdentifier_MinimumValue 	:=	136	,
	BACnetPropertyIdentifier_NotificationThreshold 	:=	137	,
	BACnetPropertyIdentifier_PreviousNotifyTime 	:=	138	,
	BACnetPropertyIdentifier_ProtocolRevision 	:=	139	,
	BACnetPropertyIdentifier_RecordsSinceNotification 	:=	140	,
	BACnetPropertyIdentifier_RecordCount 	:=	141	,
	BACnetPropertyIdentifier_StartTime 	:=	142	,
	BACnetPropertyIdentifier_StopTime 	:=	143	,
	BACnetPropertyIdentifier_StopWhenFull 	:=	144	,
	BACnetPropertyIdentifier_TotalRecordCount 	:=	145	,
	BACnetPropertyIdentifier_ValidSamples 	:=	146	,
	BACnetPropertyIdentifier_WindowInterval 	:=	147	,
	BACnetPropertyIdentifier_WindowSamples 	:=	148	,
	BACnetPropertyIdentifier_MaximumValueTimestamp 	:=	149	,
	BACnetPropertyIdentifier_MinimumValueTimestamp 	:=	150	,
	BACnetPropertyIdentifier_VarianceValue 	:=	151	,
	BACnetPropertyIdentifier_ActiveCovSubscriptions 	:=	152	,
	BACnetPropertyIdentifier_BackupFailureTimeout 	:=	153	,
	BACnetPropertyIdentifier_ConfigurationFiles 	:=	154	,
	BACnetPropertyIdentifier_DatabaseRevision 	:=	155	,
	BACnetPropertyIdentifier_DirectReading 	:=	156	,
	BACnetPropertyIdentifier_LastRestoreTime 	:=	157	,
	BACnetPropertyIdentifier_MaintenanceRequired 	:=	158	,
	BACnetPropertyIdentifier_MemberOf 	:=	159	,
	BACnetPropertyIdentifier_Mode 	:=	160	,
	BACnetPropertyIdentifier_OperationExpected 	:=	161	,
	BACnetPropertyIdentifier_Setting 	:=	162	,
	BACnetPropertyIdentifier_Silenced 	:=	163	,
	BACnetPropertyIdentifier_TrackingValue 	:=	164	,
	BACnetPropertyIdentifier_ZoneMembers 	:=	165	,
	BACnetPropertyIdentifier_LifeSafetyAlarmValues 	:=	166	,
	BACnetPropertyIdentifier_MaxSegmentsAccepted 	:=	167	,
	BACnetPropertyIdentifier_ProfileName 	:=	168	,
	BACnetPropertyIdentifier_AutoSlaveDiscovery 	:=	169	,
	BACnetPropertyIdentifier_ManualSlaveAddressBinding 	:=	170	,
	BACnetPropertyIdentifier_SlaveAddressBinding 	:=	171	,
	BACnetPropertyIdentifier_SlaveProxyEnable 	:=	172	,
	BACnetPropertyIdentifier_LastNotifyRecord 	:=	173	,
	BACnetPropertyIdentifier_ScheduleDefault 	:=	174	,
	BACnetPropertyIdentifier_AcceptedModes 	:=	175	,
	BACnetPropertyIdentifier_AdjustValue 	:=	176	,
	BACnetPropertyIdentifier_Count 	:=	177	,
	BACnetPropertyIdentifier_CountBeforeChange 	:=	178	,
	BACnetPropertyIdentifier_CountChangeTime 	:=	179	,
	BACnetPropertyIdentifier_CovPeriod 	:=	180	,
	BACnetPropertyIdentifier_InputReference 	:=	181	,
	BACnetPropertyIdentifier_LimitMonitoringInverval 	:=	182	,
	BACnetPropertyIdentifier_LoggingObject 	:=	183	,
	BACnetPropertyIdentifier_LoggingRecord 	:=	184	,
	BACnetPropertyIdentifier_Prescale 	:=	185	,
	BACnetPropertyIdentifier_PulseRate 	:=	186	,
	BACnetPropertyIdentifier_Scale 	:=	187	,
	BACnetPropertyIdentifier_ScaleFactor 	:=	188	,
	BACnetPropertyIdentifier_UpdateTime 	:=	189	,
	BACnetPropertyIdentifier_ValueBeforeChange 	:=	190	,
	BACnetPropertyIdentifier_ValueSet 	:=	191	,
	BACnetPropertyIdentifier_ValueChangeTime 	:=	192	,
	BACnetPropertyIdentifier_AlignIntervals 	:=	193	,
	BACnetPropertyIdentifier_GroupMemberNames 	:=	194	,
	BACnetPropertyIdentifier_IntervalOffset 	:=	195	,
	BACnetPropertyIdentifier_LastRestartReason 	:=	196	,
	BACnetPropertyIdentifier_LoggingType 	:=	197	,
	BACnetPropertyIdentifier_MemberStatusFlags 	:=	198	,
	BACnetPropertyIdentifier_NotificationPeriod 	:=	199	,
	BACnetPropertyIdentifier_PreviousNotifyRecord 	:=	200	,
	BACnetPropertyIdentifier_RequestedUpdateInterval 	:=	201	,
	BACnetPropertyIdentifier_RestartNotificationRecipients 	:=	202	,
	BACnetPropertyIdentifier_TimeOfDeviceRestart 	:=	203	,
	BACnetPropertyIdentifier_TimeSynchronizationInterval 	:=	204	,
	BACnetPropertyIdentifier_Trigger 	:=	205	,
	BACnetPropertyIdentifier_UTCTimeSynchronizationRecipients 	:=	206	,
	BACnetPropertyIdentifier_NodeSubtype 	:=	207	,
	BACnetPropertyIdentifier_NodeType 	:=	208	,
	BACnetPropertyIdentifier_StructuredObjectList 	:=	209	,
	BACnetPropertyIdentifier_SubordinateAnnotations 	:=	210	,
	BACnetPropertyIdentifier_SubordinateList 	:=	211	,
	BACnetPropertyIdentifier_ActualShedLevel 	:=	212	,
	BACnetPropertyIdentifier_DutyWindow 	:=	213	,
	BACnetPropertyIdentifier_ExpectedShedLevel 	:=	214	,
	BACnetPropertyIdentifier_FullDutyBaseline 	:=	215	,
	BACnetPropertyIdentifier_NodeSubtype216 	:=	216	,
	BACnetPropertyIdentifier_NodeType217 	:=	217	,
	BACnetPropertyIdentifier_RequestedShedLevel 	:=	218	,
	BACnetPropertyIdentifier_ShedDuration 	:=	219	,
	BACnetPropertyIdentifier_ShedLevelDescriptions 	:=	220	,
	BACnetPropertyIdentifier_ShedLevels 	:=	221	,
	BACnetPropertyIdentifier_StateDescription 	:=	222	,
	BACnetPropertyIdentifier_DoorAlarmState 	:=	226	,
	BACnetPropertyIdentifier_DoorExtendedPulseTime 	:=	227	,
	BACnetPropertyIdentifier_DoorMembers 	:=	228	,
	BACnetPropertyIdentifier_DoorOpenTooLongTime 	:=	229	,
	BACnetPropertyIdentifier_DoorPulseTime 	:=	230	,
	BACnetPropertyIdentifier_DoorStatus 	:=	231	,
	BACnetPropertyIdentifier_DoorUnlockDelayTime 	:=	232	,
	BACnetPropertyIdentifier_LockStatus 	:=	233	,
	BACnetPropertyIdentifier_MaskedAlarmValues 	:=	234	,
	BACnetPropertyIdentifier_SecuredStatus 	:=	235	,
	BACnetPropertyIdentifier_BackupAndRestoreState 	:=	338	,
	BACnetPropertyIdentifier_BackupPreparationTime 	:=	339	,
	BACnetPropertyIdentifier_RestoreCompletionTime 	:=	340	,
	BACnetPropertyIdentifier_RestorePreparationTime 	:=	341	,
	BACnetPropertyIdentifier_EventMessageTexts 	:=	351	,
	BACnetPropertyIdentifier_EventMessageTextsConfig 	:=	352	,
	BACnetPropertyIdentifier_ScaleOffset 	:=	512	,
	BACnetPropertyIdentifier_IoBusNr 	:=	513	,
	BACnetPropertyIdentifier_IoModuleNr 	:=	514	,
	BACnetPropertyIdentifier_IoModuleChn 	:=	515	,
	BACnetPropertyIdentifier_PersistentData 	:=	516	,
	BACnetPropertyIdentifier_CurrentlyActivePriority 	:=	517	,
	BACnetPropertyIdentifier_LastConfirmedServiceAccess 	:=	518	,
	BACnetPropertyIdentifier_DataRequestMode 	:=	519	,
	BACnetPropertyIdentifier_DataRequestCycle 	:=	520	,
	BACnetPropertyIdentifier_FileName 	:=	521
);
END_TYPE

(* Data type *)
TYPE E_BACnetRecipientChoice :
(
	BACnetRecipientChoice_device,
	BACnetRecipientChoice_address
);
END_TYPE

(* Data type *)
TYPE E_BACNETRELIABILITY:
(
	BACnetReliability_no_fault_detected :=0,
	BACnetReliability_no_sensor :=1,
	BACnetReliability_over_range :=2,
	BACnetReliability_under_range :=3,
	BACnetReliability_open_loop :=4,
	BACnetReliability_shorted_loop :=5,
	BACnetReliability_no_output :=6,
	BACnetReliability_unreliable_other :=7,
	BACnetReliability_process_error :=8,
	BACnetReliability_multi_state_fault :=9,
	BACnetReliability_configuration_error :=10,
	BACnetReliability_reserved11 :=11,
	BACnetReliability_communication_failure :=12,
	BACnetReliability_member_fault :=13
);
END_TYPE

(* Data type *)
TYPE E_BACNETSEGMENTATION:
(
	BACnetSegmentation_both :=0,
	BACnetSegmentation_transmit :=1,
	BACnetSegmentation_receive :=2,
	BACnetSegmentation_no :=3
);
END_TYPE

(* Data type *)
TYPE E_BACNETSERVICESSUPPORTEDBITS:
(
	BACnetServiceSupportedBits_AcknowledgeAlarm :=0,
	BACnetServiceSupportedBits_ConfirmedCOVNotification :=1,
	BACnetServiceSupportedBits_ConfirmedEventNotification :=2,
	BACnetServiceSupportedBits_GetAlarmSummary :=3,
	BACnetServiceSupportedBits_GetEnrollmentSummary :=4,
	BACnetServiceSupportedBits_SubscribeCOV :=5,
	BACnetServiceSupportedBits_AtomicReadFile :=6,
	BACnetServiceSupportedBits_AtomicWriteFile :=7,
	BACnetServiceSupportedBits_AddListElement :=8,
	BACnetServiceSupportedBits_RemoveListElement :=9,
	BACnetServiceSupportedBits_CreateObject :=10,
	BACnetServiceSupportedBits_DeleteObject :=11,
	BACnetServiceSupportedBits_ReadProperty :=12,
	BACnetServiceSupportedBits_ReadPropertyConditional :=13,
	BACnetServiceSupportedBits_ReadPropertyMultiple :=14,
	BACnetServiceSupportedBits_WriteProperty :=15,
	BACnetServiceSupportedBits_WritePropertyMultiple :=16,
	BACnetServiceSupportedBits_DeviceCommunicationControl :=17,
	BACnetServiceSupportedBits_ConfirmedPrivateTransfer :=18,
	BACnetServiceSupportedBits_ConfirmedTextMessage :=19,
	BACnetServiceSupportedBits_ReinitializeDevice :=20,
	BACnetServiceSupportedBits_VtOpen :=21,
	BACnetServiceSupportedBits_VtClose :=22,
	BACnetServiceSupportedBits_VtData :=23,
	BACnetServiceSupportedBits_Authenticate :=24,
	BACnetServiceSupportedBits_RequestKey :=25,
	BACnetServiceSupportedBits_IAm :=26,
	BACnetServiceSupportedBits_IHave :=27,
	BACnetServiceSupportedBits_UnconfirmedCOVNotification :=28,
	BACnetServiceSupportedBits_UnconfirmedEventNotification :=29,
	BACnetServiceSupportedBits_UnconfirmedPrivateTransfer :=30,
	BACnetServiceSupportedBits_UnconfirmedTextMessage :=31,
	BACnetServiceSupportedBits_TimeSynchronization :=32,
	BACnetServiceSupportedBits_WhoHas :=33,
	BACnetServiceSupportedBits_WhoIs :=34,
	BACnetServiceSupportedBits_ReadRange :=35,
	BACnetServiceSupportedBits_UtcTimeSynchronization :=36,
	BACnetServiceSupportedBits_LifeSafetyOperation :=37,
	BACnetServiceSupportedBits_SubscribeCOVProperty :=38,
	BACnetServiceSupportedBits_GetEventInformation :=39
);
END_TYPE

(* Data type *)
TYPE E_BACNETSILENCEDSTATE:
(
	BACnetSilencedState_unsilenced :=0,
	BACnetSilencedState_audible_silenced :=1,
	BACnetSilencedState_visible_silenced :=2,
	BACnetSilencedState_all_silenced :=3
);
END_TYPE

(* Data type *)
TYPE E_BACnetSpecialEventChoice :
(
(*
	enum BACnetSpecialEventChoice
	{
	      calendarEntry,
	      calendarReference,
	      MaxBACnetSpecialEventChoice
	};
*)
	BACnetSpecialEventChoice_calendarEntry,
	BACnetSpecialEventChoice_calendarReference
);
END_TYPE

(* Data type *)
TYPE E_BACNETSTATUSFLAGS:
(
	BACnetStatusFlags_in_alarm :=0,
	BACnetStatusFlags_fault :=1,
	BACnetStatusFlags_overridden :=2,
	BACnetStatusFlags_out_of_service :=3
);
END_TYPE

(* Data type *)
TYPE E_BACNETSTRINGENCODINGTYPES :
(
	BACnetStringEncodingTypes_AnsiUtf8	:= 0,
	BACnetStringEncodingTypes_DBCS		:= 1,
	BACnetStringEncodingTypes_JIS		:= 2,
	BACnetStringEncodingTypes_UCS4		:= 3,
	BACnetStringEncodingTypes_UCS2		:= 4,
	BACnetStringEncodingTypes_ISO8859	:= 5
);
END_TYPE

(*
---------------------------------------------
ISO8859
---------------------------------------------
Part 1	Latin-1
 Western European
Part 2	Latin-2
 Central European
Part 3	Latin-3
 South European
Part 4	Latin-4
 North European
Part 5	Latin/Cyrillic
Part 6	Latin/Arabic
Part 7	Latin/Greek
Part 8	Latin/Hebrew
Part 9	Latin-5 
Turkish
Part 10	Latin-6 
Nordic
Part 11	Latin/Thai
Part 12	"non-existent part" Latin/Devanagari
Part 13	Latin-7
 Baltic Rim
Part 14	Latin-8
 Celtic
Part 15	Latin-9
Part 16	Latin-10
 South-Eastern European
---------------------------------------------
*)

(* Data type *)
TYPE E_BACnetTimeStampChoice :
(
	BACnetTimeStampChoice_ts_time,
    BACnetTimeStampChoice_sequenceNumber,
    BACnetTimeStampChoice_dateTime
);
END_TYPE

(* Data type *)
TYPE E_BACNETUNIT:
(
	BACnetUnit_Area_square_meters	:=	0	,
	BACnetUnit_Area_square_feet	:=	1	,
	BACnetUnit_Electrical_milliamperes	:=	2	,
	BACnetUnit_Electrical_amperes	:=	3	,
	BACnetUnit_Electrical_ohms	:=	4	,
	BACnetUnit_Electrical_volts	:=	5	,
	BACnetUnit_Electrical_kilovolts	:=	6	,
	BACnetUnit_Electrical_megavolts	:=	7	,
	BACnetUnit_Electrical_volt_amperes	:=	8	,
	BACnetUnit_Electrical_kilovolt_amperes	:=	9	,
	BACnetUnit_Electrical_megavolt_amperes	:=	10	,
	BACnetUnit_Electrical_volt_amperes_reactive	:=	11	,
	BACnetUnit_Electrical_kilovolt_amperes_reactive	:=	12	,
	BACnetUnit_Electrical_megavolt_amperes_reactive	:=	13	,
	BACnetUnit_Electrical_degrees_phase	:=	14	,
	BACnetUnit_Electrical_power_factor	:=	15	,
	BACnetUnit_Energy_joules	:=	16	,
	BACnetUnit_Energy_kilojoules	:=	17	,
	BACnetUnit_Energy_watt_hours	:=	18	,
	BACnetUnit_Energy_kilowatt_hours	:=	19	,
	BACnetUnit_Energy_btus	:=	20	,
	BACnetUnit_Energy_therms	:=	21	,
	BACnetUnit_Energy_ton_hours	:=	22	,
	BACnetUnit_Enthalpy_joules_per_kilogram_dry_air	:=	23	,
	BACnetUnit_Enthalpy_btus_per_pound_dry_air	:=	24	,
	BACnetUnit_Frequency_cycles_per_hour	:=	25	,
	BACnetUnit_Frequency_cycles_per_minute	:=	26	,
	BACnetUnit_Frequency_hertz	:=	27	,
	BACnetUnit_Humidity_grams_of_water_per_kilogram_dry_air	:=	28	,
	BACnetUnit_Humidity_percent_relative_humidity	:=	29	,
	BACnetUnit_Length_millimeters	:=	30	,
	BACnetUnit_Length_meters	:=	31	,
	BACnetUnit_Length_inches	:=	32	,
	BACnetUnit_Length_feet	:=	33	,
	BACnetUnit_Light_watts_per_square_foot	:=	34	,
	BACnetUnit_Light_watts_per_square_meter	:=	35	,
	BACnetUnit_Light_lumens	:=	36	,
	BACnetUnit_Light_luxes	:=	37	,
	BACnetUnit_Light_foot_candles	:=	38	,
	BACnetUnit_Mass_kilograms	:=	39	,
	BACnetUnit_Mass_pounds_mass	:=	40	,
	BACnetUnit_Mass_tons	:=	41	,
	BACnetUnit_MassFlow_kilograms_per_second	:=	42	,
	BACnetUnit_MassFlow_kilograms_per_minute	:=	43	,
	BACnetUnit_MassFlow_kilograms_per_hour	:=	44	,
	BACnetUnit_MassFlow_pounds_mass_per_minute	:=	45	,
	BACnetUnit_MassFlow_pounds_mass_per_hour	:=	46	,
	BACnetUnit_Power_watts	:=	47	,
	BACnetUnit_Power_kilowatts	:=	48	,
	BACnetUnit_Power_megawatts	:=	49	,
	BACnetUnit_Power_btus_per_hour	:=	50	,
	BACnetUnit_Power_horsepower	:=	51	,
	BACnetUnit_Power_tons_refrigeration	:=	52	,
	BACnetUnit_Pressure_pascals	:=	53	,
	BACnetUnit_Pressure_kilopascals	:=	54	,
	BACnetUnit_Pressure_bars	:=	55	,
	BACnetUnit_Pressure_pounds_force_per_square_inch	:=	56	,
	BACnetUnit_Pressure_centimeters_of_water	:=	57	,
	BACnetUnit_Pressure_inches_of_water	:=	58	,
	BACnetUnit_Pressure_millimeters_of_mercury	:=	59	,
	BACnetUnit_Pressure_centimeters_of_mercury	:=	60	,
	BACnetUnit_Pressure_inches_of_mercury	:=	61	,
	BACnetUnit_Temperature_degrees_Celsius	:=	62	,
	BACnetUnit_Temperature_degrees_Kelvin	:=	63	,
	BACnetUnit_Temperature_degrees_Fahrenheit	:=	64	,
	BACnetUnit_Temperature_degree_days_Celsius	:=	65	,
	BACnetUnit_Temperature_degree_days_Fahrenheit	:=	66	,
	BACnetUnit_Time_years	:=	67	,
	BACnetUnit_Time_months	:=	68	,
	BACnetUnit_Time_weeks	:=	69	,
	BACnetUnit_Time_days	:=	70	,
	BACnetUnit_Time_hours	:=	71	,
	BACnetUnit_Time_minutes	:=	72	,
	BACnetUnit_Time_seconds	:=	73	,
	BACnetUnit_Velocity_meters_per_second	:=	74	,
	BACnetUnit_Velocity_kilometers_per_hour	:=	75	,
	BACnetUnit_Velocity_feet_per_second	:=	76	,
	BACnetUnit_Velocity_feet_per_minute	:=	77	,
	BACnetUnit_Velocity_miles_per_hour	:=	78	,
	BACnetUnit_Volume_cubic_feet	:=	79	,
	BACnetUnit_Volume_cubic_meters	:=	80	,
	BACnetUnit_Volume_imperial_gallons	:=	81	,
	BACnetUnit_Volume_liters	:=	82	,
	BACnetUnit_Volume_us_gallons	:=	83	,
	BACnetUnit_VolumetricFlow_cubic_feet_per_minute	:=	84	,
	BACnetUnit_VolumetricFlow_cubic_meters_per_second	:=	85	,
	BACnetUnit_VolumetricFlow_imperial_gallons_per_minute	:=	86	,
	BACnetUnit_VolumetricFlow_liters_per_second	:=	87	,
	BACnetUnit_VolumetricFlow_liters_per_minute	:=	88	,
	BACnetUnit_VolumetricFlow_us_gallons_per_minute	:=	89	,
	BACnetUnit_Other_degrees_angular	:=	90	,
	BACnetUnit_Other_degrees_Celsius_per_hour	:=	91	,
	BACnetUnit_Other_degrees_Celsius_per_minute	:=	92	,
	BACnetUnit_Other_degrees_Fahrenheit_per_hour	:=	93	,
	BACnetUnit_Other_degrees_Fahrenheit_per_minute	:=	94	,
	BACnetUnit_Other_no_units	:=	95	,
	BACnetUnit_Other_parts_per_million	:=	96	,
	BACnetUnit_Other_parts_per_billion	:=	97	,
	BACnetUnit_Other_percent	:=	98	,
	BACnetUnit_Other_percent_per_second	:=	99	,
	BACnetUnit_Other_per_minute	:=	100	,
	BACnetUnit_Other_per_second	:=	101	,
	BACnetUnit_Other_psi_per_degree_Fahrenheit	:=	102	,
	BACnetUnit_Other_radians	:=	103	,
	BACnetUnit_Other_revolutions_per_minute	:=	104	,
	BACnetUnit_Currency_currency1	:=	105	,
	BACnetUnit_Currency_currency2	:=	106	,
	BACnetUnit_Currency_currency3	:=	107	,
	BACnetUnit_Currency_currency4	:=	108	,
	BACnetUnit_Currency_currency5	:=	109	,
	BACnetUnit_Currency_currency6	:=	110	,
	BACnetUnit_Currency_currency7	:=	111	,
	BACnetUnit_Currency_currency8	:=	112	,
	BACnetUnit_Currency_currency9	:=	113	,
	BACnetUnit_Currency_currency10	:=	114	,
	BACnetUnit_Area_square_inches	:=	115	,
	BACnetUnit_Area_square_centimeters	:=	116	,
	BACnetUnit_Enthalpy_btus_per_pound	:=	117	,
	BACnetUnit_Length_centimeters	:=	118	,
	BACnetUnit_MassFlow_pounds_mass_per_second	:=	119	,
	BACnetUnit_Temperature_delta_degrees_Fahrenheit	:=	120	,
	BACnetUnit_Temperature_delta_degrees_Kelvin	:=	121	,
	BACnetUnit_Electrical_kilohms	:=	122	,
	BACnetUnit_Electrical_megohms	:=	123	,
	BACnetUnit_Electrical_millivolts	:=	124	,
	BACnetUnit_Energy_kilojoules_per_kilogram	:=	125	,
	BACnetUnit_Energy_megajoules	:=	126	,
	BACnetUnit_Entropy_joules_per_degree_Kelvin	:=	127	,
	BACnetUnit_Entropy_joules_per_kilogram_degree_Kelvin	:=	128	,
	BACnetUnit_Frequency_kilohertz	:=	129	,
	BACnetUnit_Frequency_megahertz	:=	130	,
	BACnetUnit_Frequency_per_hour	:=	131	,
	BACnetUnit_Power_milliwatts	:=	132	,
	BACnetUnit_Pressure_hectopascals	:=	133	,
	BACnetUnit_Pressure_millibars	:=	134	,
	BACnetUnit_VolumetricFlow_cubic_meters_per_hour	:=	135	,
	BACnetUnit_VolumetricFlow_liters_per_hour	:=	136	,
	BACnetUnit_Other_kilowatt_hours_per_square_meter	:=	137	,
	BACnetUnit_Other_kilowatt_hours_per_square_foot	:=	138	,
	BACnetUnit_Other_megajoules_per_square_meter	:=	139	,
	BACnetUnit_Other_megajoules_per_square_foot	:=	140	,
	BACnetUnit_Other_watts_per_square_meter_degree_kelvin	:=	141	,
	BACnetUnit_VolumetricFlow_cubic_feet_per_second	:=	142	,
	BACnetUnit_Other_percent_obscuration_per_foot	:=	143	,
	BACnetUnit_Other_percent_obscuration_per_meter	:=	144	,
	BACnetUnit_Electrical_milliohms	:=	145	,
	BACnetUnit_Energy_megawatt_hours	:=	146	,
	BACnetUnit_Energy_kilo_btus	:=	147	,
	BACnetUnit_Energy_mega_btus	:=	148	,
	BACnetUnit_Enthalpy_kilojoules_per_kilogram_dry_air	:=	149	,
	BACnetUnit_Enthalpy_megajoules_per_kilogram_dry_air	:=	150	,
	BACnetUnit_Entropy_kilojoules_per_degree_Kelvin	:=	151	,
	BACnetUnit_Entropy_megajoules_per_degree_Kelvin	:=	152	,
	BACnetUnit_Force_newton	:=	153	,
	BACnetUnit_MassFlow_grams_per_second	:=	154	,
	BACnetUnit_MassFlow_grams_per_minute	:=	155	,
	BACnetUnit_MassFlow_tons_per_hour	:=	156	,
	BACnetUnit_Power_kilo_btus_per_hour	:=	157	,
	BACnetUnit_Time_hundredths_seconds	:=	158	,
	BACnetUnit_Time_milliseconds	:=	159	,
	BACnetUnit_Torque_newton_meters	:=	160	,
	BACnetUnit_Velocity_millimeters_per_second	:=	161	,
	BACnetUnit_Velocity_millimeters_per_minute	:=	162	,
	BACnetUnit_Velocity_meters_per_minute	:=	163	,
	BACnetUnit_Velocity_meters_per_hour	:=	164	,
	BACnetUnit_VolumetricFlow_cubic_meters_per_minute	:=	165	,
	BACnetUnit_Acceleration_meters_per_second_per_second	:=	166	,
	BACnetUnit_Electrical_amperes_per_meter	:=	167	,
	BACnetUnit_Electrical_amperes_per_square_meter	:=	168	,
	BACnetUnit_Electrical_ampere_square_meters	:=	169	,
	BACnetUnit_Electrical_farads	:=	170	,
	BACnetUnit_Electrical_henrys	:=	171	,
	BACnetUnit_Electrical_ohm_meters	:=	172	,
	BACnetUnit_Electrical_siemens	:=	173	,
	BACnetUnit_Electrical_siemens_per_meter	:=	174	,
	BACnetUnit_Electrical_teslas	:=	175	,
	BACnetUnit_Electrical_volts_per_degree_Kelvin	:=	176	,
	BACnetUnit_Electrical_volts_per_meter	:=	177	,
	BACnetUnit_Electrical_webers	:=	178	,
	BACnetUnit_Light_candelas	:=	179	,
	BACnetUnit_Light_candelas_per_square_meter	:=	180	,
	BACnetUnit_Temperature_degrees_Kelvin_per_hour	:=	181	,
	BACnetUnit_Temperature_degrees_Kelvin_per_minute	:=	182	,
	BACnetUnit_Other_joule_seconds	:=	183	,
	BACnetUnit_Other_radians_per_second	:=	184	,
	BACnetUnit_Other_square_meters_per_Newton	:=	185	,
	BACnetUnit_Other_kilograms_per_cubic_meter	:=	186	,
	BACnetUnit_Other_newton_seconds	:=	187	,
	BACnetUnit_Other_newtons_per_meter	:=	188	,
	BACnetUnit_Other_watts_per_meter_per_degree_Kelvin	:=	189	,
	BACnetUnit_micro_siemens	:=	190	,
	BACnetUnit_cubic_feet_per_hour	:=	191	,
	BACnetUnit_us_gallons_per_hour	:=	192	,
	BACnetUnit_kilometers	:=	193	,
	BACnetUnit_micrometers	:=	194	,
	BACnetUnit_grams	:=	195	,
	BACnetUnit_milligrams	:=	196	,
	BACnetUnit_milliliters	:=	197	,
	BACnetUnit_milliliters_per_second	:=	198	,
	BACnetUnit_decibels	:=	199	,
	BACnetUnit_decibels_millivolt	:=	200	,
	BACnetUnit_decibels_volt	:=	201	,
	BACnetUnit_millisiemens	:=	202	,
	BACnetUnit_watt_hours_reactive	:=	203	,
	BACnetUnit_kilowatt_hours_reactive	:=	204	,
	BACnetUnit_megawatt_hours_reactive	:=	205	,
	BACnetUnit_millimeters_of_water	:=	206	,
	BACnetUnit_per_mille	:=	207	,
	BACnetUnit_grams_per_gram	:=	208	,
	BACnetUnit_kilograms_per_kilogram	:=	209	,
	BACnetUnit_grams_per_kilogram	:=	210	,
	BACnetUnit_milligrams_per_gram	:=	211	,
	BACnetUnit_milligrams_per_kilogram	:=	212	,
	BACnetUnit_grams_per_milliliter	:=	213	,
	BACnetUnit_grams_per_liter	:=	214	,
	BACnetUnit_milligrams_per_liter	:=	215	,
	BACnetUnit_micrograms_per_liter	:=	216	,
	BACnetUnit_grams_per_cubic_meter	:=	217	,
	BACnetUnit_milligrams_per_cubic_meter	:=	218	,
	BACnetUnit_micrograms_per_cubic_meter	:=	219	,
	BACnetUnit_nanograms_per_cubic_meter	:=	220	,
	BACnetUnit_grams_per_cubic_centimeter	:=	221	,
	BACnetUnit_becquerels	:=	222	,
	BACnetUnit_kilobecquerels	:=	223	,
	BACnetUnit_megabecquerels	:=	224	,
	BACnetUnit_gray	:=	225	,
	BACnetUnit_milligray	:=	226	,
	BACnetUnit_microgray	:=	227	,
	BACnetUnit_sieverts	:=	228	,
	BACnetUnit_millisieverts	:=	229	,
	BACnetUnit_microsieverts	:=	230	,
	BACnetUnit_microsieverts_per_hour	:=	231	,
	BACnetUnit_decibels_a	:=	232	,
	BACnetUnit_nephelometric_turbidity_unit	:=	233	,
	BACnetUnit_pH	:=	234	,
	BACnetUnit_grams_per_square_meter	:=	235	,
	BACnetUnit_minutes_per_degree_kelvin	:=	236
);
END_TYPE

(* Data type *)
TYPE FB_BACnet_Accumulator_R9 : FB_BACnet_Accumulator;
END_TYPE

(* Data type *)
TYPE FB_BACnet_AnalogInput_R9 : FB_BACnet_AnalogInput;
END_TYPE

(* Data type *)
TYPE FB_BACnet_AnalogOutput_R9 : FB_BACnet_AnalogOutput;
END_TYPE

(* Data type *)
TYPE FB_BACnet_AnalogValue_R9 : FB_BACnet_AnalogValue;
END_TYPE

(* Data type *)
TYPE FB_BACnet_Averaging_R9 : FB_BACnet_Averaging;
END_TYPE

(* Data type *)
TYPE FB_BACnet_BinaryInput_R9 : FB_BACnet_BinaryInput;
END_TYPE

(* Data type *)
TYPE FB_BACnet_BinaryOutput_R9 : FB_BACnet_BinaryOutput;
END_TYPE

(* Data type *)
TYPE FB_BACnet_BinaryValue_R9 : FB_BACnet_BinaryValue;
END_TYPE

(* Data type *)
TYPE FB_BACnet_Calendar_R9 : FB_BACnet_Calendar;
END_TYPE

(* Data type *)
TYPE FB_BACnet_Command_R9 : FB_BACnet_Command;
END_TYPE

(* Data type *)
TYPE FB_BACnet_Device_R9 : FB_BACnet_Device;
END_TYPE

(* Data type *)
TYPE FB_BACnet_EventEnrollment_R9 : FB_BACnet_EventEnrollment;
END_TYPE

(* Data type *)
TYPE FB_BACnet_File_R9 : FB_BACnet_File;
END_TYPE

(* Data type *)
TYPE FB_BACnet_Group_R9 : FB_BACnet_Group;
END_TYPE

(* Data type *)
TYPE FB_BACnet_Loop_R9 : FB_BACnet_Loop;
END_TYPE

(* Data type *)
TYPE FB_BACnet_MultiStateInput_R9 : FB_BACnet_MultiStateInput;
END_TYPE

(* Data type *)
TYPE FB_BACnet_MultiStateOutput_R9 : FB_BACnet_MultiStateOutput;
END_TYPE

(* Data type *)
TYPE FB_BACnet_MultiStateValue_R9 : FB_BACnet_MultiStateValue;
END_TYPE

(* Data type *)
TYPE FB_BACnet_NotificationClass_R9 : FB_BACnet_NotificationClass;
END_TYPE

(* Data type *)
TYPE FB_BACnet_Program_R9 : FB_BACnet_Program;
END_TYPE

(* Data type *)
TYPE FB_BACnet_PulseConverter_R9 : FB_BACnet_PulseConverter;
END_TYPE

(* Data type *)
TYPE FB_BACnet_Schedule_R9 : FB_BACnet_Schedule;
END_TYPE

(* Data type *)
TYPE FB_BACnet_TrendLog_R9 : FB_BACnet_TrendLog;
END_TYPE

(* Data type *)
TYPE ST_BACnet_AdsConnection :
STRUCT
	bValid		: BOOL; (* information are valid *)
	nReload		: USINT; (* reload counter *)
	sAmsNetId	: T_AmsNetId;
	nAmsPort	: T_AmsPort := 1000;
	bServer		: BOOL;
	bClient		: BOOL;
	bNSink		: BOOL;
	nDeviceId	: UDINT; (* Device object instance resp. BACnet ID *)
END_STRUCT
END_TYPE

(* Data type *)
TYPE ST_BACnet_CalendarEntryDate :
STRUCT
(*
	typedef struct _BACnetCalendarEntry
	{
	      BACnetCalendarEntryChoice choice;
	      union
	      {
	            BACnetDate              date;
	            BACnetDateRange   dateRange;
	            BACnetWeekNDay          weekNDay;
	      };
	}BACnetCalendarEntry, *PBACnetCalendarEntry;
*)
	eEntryChoice		: E_BACnetCalendarEntryChoice;
	nRes				: WORD; (* ENUM alignment *)
	stDate				: ST_BACnet_Date;
END_STRUCT
END_TYPE

(* Data type *)
TYPE ST_BACnet_CalendarEntryDateRange :
STRUCT
(*
	typedef struct _BACnetCalendarEntry
	{
	      BACnetCalendarEntryChoice choice;
	      union
	      {
	            BACnetDate              date;
	            BACnetDateRange   dateRange;
	            BACnetWeekNDay          weekNDay;
	      };
	}BACnetCalendarEntry, *PBACnetCalendarEntry;
*)
	eEntryChoice		: E_BACnetCalendarEntryChoice;
	nRes				: WORD; (* ENUM alignment *)
	stStartDate			: ST_BACnet_Date;
	stEndDate			: ST_BACnet_Date;
END_STRUCT
END_TYPE

(* Data type *)
TYPE ST_BACnet_CalendarEntryWeekNDay :
STRUCT
(*
	typedef struct _BACnetCalendarEntry
	{
	      BACnetCalendarEntryChoice choice;
	      union
	      {
	            BACnetDate              date;
	            BACnetDateRange   dateRange;
	            BACnetWeekNDay          weekNDay;
	      };
	}BACnetCalendarEntry, *PBACnetCalendarEntry;
*)
	eEntryChoice	: E_BACnetCalendarEntryChoice;
	nRes1			: WORD; (* ENUM alignment *)
	iMonth			: USINT;
	iWeekOfMonth	: USINT;
	iDay			: USINT;
	nRes2			: USINT; (* weekNDay alignment *)
END_STRUCT
END_TYPE

(* Data type *)
TYPE ST_BACnet_CharacterStringExt :
STRUCT
	cookie		: BYTE; (* 0 -> DO differentiate normal strings *)
	encoding	: BYTE;
	strLen		: UINT;
	stringData	: ARRAY[1..BACnet_STRING_MAXLENGTH] OF BYTE;
END_STRUCT
END_TYPE

(* Data type *)
TYPE ST_BACnet_CharacterStringExtListEntry :
STRUCT
(* list header *)
	nEntrySize	: DWORD; (* byte size of data *)
	hdrInfo		: DWORD;
(* data *)
	extString	: ST_BACnet_CharacterStringExt;
END_STRUCT
END_TYPE

(* Data type *)
TYPE ST_BACnet_ConfirmedServiceDiag :
STRUCT
	nReqSend: DWORD; (* ULONG *)
	nReqSendFail: DWORD; (* ULONG *)
	nReqRecv: DWORD; (* ULONG *)
	nReqRecvFail: DWORD; (* ULONG *)
	nAckSend: DWORD; (* ULONG *)
	nAckSendFail: DWORD; (* ULONG *)
	nAckRecv: DWORD; (* ULONG *)
	nAckRecvFail: DWORD; (* ULONG *)
END_STRUCT
END_TYPE

(* Data type *)
TYPE ST_BACnet_DailySchedule :
STRUCT
(*
	PropWeeklySchedule:
	
	typedef struct _BACnetDailySchedule
	{
	      DWORD nEntrySize; // 0x80000000 -> next entry
	      DWORD reserved;
	      BACnetTimeValueList listEntry;
	} BACnetDailySchedule, *PBACnetDailySchedule;
*)
	nEntrySize	: DWORD;
	nRes		: DWORD;
	stListEntry	: ST_BACnet_TimeValueList;
END_STRUCT
END_TYPE

(* Data type *)
TYPE ST_BACnet_Date :
STRUCT
	nYear		: BYTE := 16#FF; (* year minus 1900 X'FF' = unspecified *)
	nMonth		: BYTE := 16#FF; (* (1.. 12) 1 = January X'FF' = unspecified *)
	nDay		: BYTE := 16#FF;	(* day OF month (1..31), X'FF' = unspecified *)
	nDayOfWeek	: BYTE := 16#FF;	(* day OF week (1..7) 1 = Monday -- 7 = Sunday -- X'FF' = unspecified *)
END_STRUCT
END_TYPE

(* Data type *)
TYPE ST_BACnet_DateTime :
STRUCT
	stDate		: ST_BACnet_Date;
	stTime		: ST_BACnet_Time;
END_STRUCT
END_TYPE

(* Data type *)
TYPE ST_BACnet_DestinationDevice :
STRUCT
	nValidDaysFlags	: DWORD; (* Bit: 9 = Sunday, 10 = Saturday, 11 = Friday, 12 = Thursday, 13 = Wednesday, 14 = Tuesday, 15 = Monday *)
	stFromTime		: ST_BACnet_Time;
	stToTime		: ST_BACnet_Time;
	stRecipient		: ST_BACnet_RecipientDevice;
	res1			: ARRAY[0..11] OF BYTE; (* allignment *)
	nProcessId		: UDINT;
	nEventTransBits	: DWORD; (* Bit: 12 = to_offnormal, 13 = to_fault, 14 = to_normal *)
	bIssueConfNot	: BOOL;
	res2			: ARRAY[0..2] OF BYTE; (* allignment *)
END_STRUCT
END_TYPE

(* Data type *)
TYPE ST_BACnet_DiagEthStatistics :
STRUCT
	ethStat: ST_BACnet_TcIoEthStatistic;
	txRxErrCnt: ST_BACnet_TcIoEthTxRxErrorCount;
END_STRUCT
END_TYPE

(* Data type *)
TYPE ST_BACnet_Diagnosis :
STRUCT
	ethDevice: ST_BACnet_DiagEthStatistics;
	execTiming: ST_BACnet_DiagnosisTiming;
	frameStatistics: ST_BACnet_FrameStatistics;
	nRes1 : DWORD;
	info: ST_BACnet_Info;
	nRes2 : DWORD;
	serverInfo: ST_BACnet_ServerStatistics;
	lastUpdate: ST_BACnet_DateTime;
	nRes3 : DWORD;
END_STRUCT
END_TYPE

(* Data type *)
TYPE ST_BACnet_DiagnosisTiming :
STRUCT
	msIoInCurExecutionTime: DWORD; (* ULONG *)
	msIoInMinExecutionTime: DWORD; (* ULONG *)
	msIoInMaxExecutionTime: DWORD; (* ULONG *)
	msIoOutCurExecutionTime: DWORD; (* ULONG *)
	msIoOutMinExecutionTime: DWORD; (* ULONG *)
	msIoOutMaxExecutionTime: DWORD; (* ULONG *)
	msCycleCurExecutionTime: DWORD; (* ULONG *)
	msCycleMinExecutionTime: DWORD; (* ULONG *)
	msCycleMaxExecutionTime: DWORD; (* ULONG *)
	msInputCurDistanceTime: DWORD; (* ULONG *)
	msInputMinDistanceTime: DWORD; (* ULONG *)
	msInputMaxDistanceTime: DWORD; (* ULONG *)
END_STRUCT
END_TYPE

(* Data type *)
TYPE ST_BACnet_EventTransitionBits:
STRUCT
	to_offnormal : BOOL;
	to_fault : BOOL;
	to_normal : BOOL;
END_STRUCT
END_TYPE

(* Data type *)
TYPE ST_BACnet_ExceptionScheduleBool :
STRUCT
	bReqGet		: BOOL; (* set TRUE if property should reloaded, TRUE --> FALSE = request accepted (starting reload) *)
	bReqSet		: BOOL; (* set TRUE for property write request, TRUE --> FALSE = request accepted (starting storage) *)
	nGet		: USINT; (* reload counter, count up if property was loaded successful *)
	nSet		: USINT; (* save counter, count up if property was stored successful *)
	bBusy		: BOOL; (* started writing data into "arrEntries", don't write data to avoid concurrent access *)
	arrEntries	: ARRAY[0..BACnet_MaxExSchEntries] OF ST_BACnet_ExceptionScheduleEntryBool;
END_STRUCT
END_TYPE

(* Data type *)
TYPE ST_BACnet_ExceptionScheduleCalDate :
STRUCT
	stStart			: ST_BACnet_Date;
	stEnd			: ST_BACnet_Date;
END_STRUCT
END_TYPE

(* Data type *)
TYPE ST_BACnet_ExceptionScheduleCalRef :
STRUCT
	tCalObjectId	: T_BACnet_ObjectIdentifier := 16#FFFFFFFF;
END_STRUCT
END_TYPE

(* Data type *)
TYPE ST_BACnet_ExceptionScheduleCalWnD :
STRUCT
	iMonth			: USINT; (* 255 = all months of year *)
	iWeekOfMonth	: USINT; (* 255 = all weeks of month *)
	iDay			: USINT; (* 255 = all days of month *)
END_STRUCT
END_TYPE

(* Data type *)
TYPE ST_BACnet_ExceptionScheduleEntryBool :
STRUCT
	eEntryType		: E_BACnetCalendarEntryType;
	ePriority		: E_BACnetPriority;
	stDate			: ST_BACnet_ExceptionScheduleCalDate; (* date / date range *)
	stWeekNDay		: ST_BACnet_ExceptionScheduleCalWnD; (* week and day *)
	stCalRef		: ST_BACnet_ExceptionScheduleCalRef; (* week and day *)
	arrTimeValue	: ARRAY[0..BACnet_MaxTimeValues] OF ST_BACnet_TimeValueBool;
END_STRUCT
END_TYPE

(* Data type *)
TYPE ST_BACnet_ExceptionScheduleEntryReal :
STRUCT
	eEntryType		: E_BACnetCalendarEntryType;
	ePriority		: E_BACnetPriority;
	stDate			: ST_BACnet_ExceptionScheduleCalDate; (* date / date range *)
	stWeekNDay		: ST_BACnet_ExceptionScheduleCalWnD; (* week and day *)
	stCalRef		: ST_BACnet_ExceptionScheduleCalRef; (* week and day *)
	arrTimeValue	: ARRAY[0..BACnet_MaxTimeValues] OF ST_BACnet_TimeValueReal;
END_STRUCT
END_TYPE

(* Data type *)
TYPE ST_BACnet_ExceptionScheduleReal :
STRUCT
	bReqGet		: BOOL; (* set TRUE if property should reloaded, TRUE --> FALSE = request accepted (starting reload) *)
	bReqSet		: BOOL; (* set TRUE for property write request, TRUE --> FALSE = request accepted (starting storage) *)
	nGet		: USINT; (* reload counter, count up if property was loaded successful *)
	nSet		: USINT; (* save counter, count up if property was stored successful *)
	bBusy		: BOOL; (* started writing data into "arrEntries", don't write data to avoid concurrent access *)
	arrEntries	: ARRAY[0..BACnet_MaxExSchEntries] OF ST_BACnet_ExceptionScheduleEntryReal;
END_STRUCT
END_TYPE

(* Data type *)
TYPE ST_BACnet_FrameStatistics :
STRUCT
	confirmed: ARRAY[0..29] OF ST_BACnet_ConfirmedServiceDiag; (* [SERVICE_CONFIRMED_MAX + 1]; 29 + 1 *)
	unConfirmed: ARRAY[0..9] OF ST_BACnet_UnConfirmedServiceDiag; (* [SERVICE_UNCONFIRMED_MAX + 1]; 9 *)
	nSegmSendTimeouts: DWORD; (* ULONG *)
	nFrameAllocFailCnt: DWORD; (* ULONG *)
	nFrameSendCnt: DWORD; (* ULONG *)
	nFrameSendFailCnt: DWORD; (* ULONG *)
	nFrameRecvCnt: DWORD; (* ULONG *)
	nFrameRecvFailCnt: DWORD; (* ULONG *)
	nLinkStatusChangedCnt: DWORD; (* ULONG *)
END_STRUCT
END_TYPE

(* Data type *)
TYPE ST_BACnet_GlobalAdsBuffer :
STRUCT
	bTestSet	: BOOL;
	iLocked		: DINT; (* -1 Buffer not ready, 0 Buffer ready, 1..n Buffer used (locked) *)
	arrData		: ARRAY[0..BACnet_ADSBufferSize] OF BYTE;
END_STRUCT
END_TYPE

(* Data type *)
TYPE ST_BACnet_Info :
STRUCT
	nAmsAllocCnt: DINT; (* LONG *)
	nAmsAllocCntMax: DWORD; (* ULONG *)
	nAmsAllocFailCnt: DWORD; (* ULONG *)
	nAvailPhysMemBytes: DWORD; (* ULONG *)
	nAvailFlashMemBytes: ARRAY[0..1] OF DWORD; (* ULONGLONG *)
	nRecvFrameFifoSize: DWORD; (* ULONG *)
	nEmptyFrameFifoSize: DWORD; (* ULONG *)
	nRecvSegmUDPFramesListSize: DWORD; (* ULONG *)
	nRecvSegmFramesListSize: DWORD; (* ULONG *)
	nSendSegmFramesListSize: DWORD; (* ULONG *)
	nClientScanListSize: DWORD; (* ULONG *)
	nAmsRecvMissCount: DWORD; (* ULONG *)
END_STRUCT
END_TYPE

(* Data type *)
TYPE ST_BACnet_LimitEnable:
STRUCT
	lowLimitEnable : BOOL;
	highLimitEnable : BOOL;
END_STRUCT
END_TYPE

(* Data type *)
TYPE ST_BACnet_LogBufferEntryReal :
STRUCT
	nTimeStamp	: DWORD; (* 100ms since 1900 *)
	stDateTime	: ST_BACnet_DateTime; (* BACnet time stamp *)
	fValue		: REAL;
END_STRUCT
END_TYPE

(* Data type *)
TYPE ST_BACnet_LogBufferReal :
STRUCT
	nGet		: USINT; (* Update date counter *)
	sObjectDesc	: T_MAXSTRING; (* Object description *)
	nCount		: UDINT; (* log buffer entries *)
	arrEntries	: ARRAY[0..BACnet_MaxLogBufferEntries] OF ST_BACnet_LogBufferEntryReal;
END_STRUCT
END_TYPE

(* Data type *)
TYPE ST_BACnet_LogDatum :
STRUCT
(*

typedef struct _BACnetLogDatum
{
      BACnetLogRecordChoice choice;
      union
      {
            DWORD logStatus; // BitString ... of type BACnetLogStatus
            BOOL booleanValue;
            FLOAT realValue;
            EnumerationValueType enumerationValue;
            ULONG unsignedValue;
            DWORD signedValue;
            DWORD bitstringValue;
            DWORD nullValue;
            BACnetError failure; 
            FLOAT timeChange;
            AnyType anyValue; // ABSTRACT-SYNTAX.&Type
      };
}BACnetLogDatum, *PBACnetLogDatum;

*)
	choice	: E_BACnetLogRecordChoice;
	nRes	: WORD; (* ENUM alignment to 4 byte *)
	nData	: ARRAY[0..4] OF DWORD; (* 20 byte min. size - data type depending on choice selection *)
END_STRUCT
END_TYPE

(* Data type *)
TYPE ST_BACnet_LogDatumList :
STRUCT
(*

typedef struct _BACnetLogDatumList
{
      DWORD nEntrySize; // 0x80000000 -> next entry
      DWORD reserved;
      BACnetLogDatum listEntry;
}BACnetLogDatumList, *PBACnetLogDatumList;

*)
	nEntrySize	: DWORD; (* 0x80000000 -> next entry *)
	reserved	: DWORD;
	listEntry	: ST_BACnet_LogDatum; (* first entry of log datum list *)
END_STRUCT
END_TYPE

(* Data type *)
TYPE ST_BACnet_LogRecord :
STRUCT
(*

typedef STRUCT _BACnetLogRecord
{
      ULONG validFields;
      BACnetDateTime timestamp;          // [0]
      DWORD statusFlags;                       // [2] optional
      BACnetLogDatumList logDatum;  // [1]
}BACnetLogRecord, *PBACnetLogRecord;

*)
	validFields	: UDINT;
	timestamp	: ST_BACnet_DateTime;
	statusFlags	: DWORD;
	logDatum	: ST_BACnet_LogDatumList;
END_STRUCT
END_TYPE

(* Data type *)
TYPE ST_BACnet_LogRecordList :
STRUCT
(*

typedef struct _BACnetLogRecordList
{
      DWORD nEntrySize; // 0x80000000 -> next entry
      DWORD nSequence;  // "reserved"     -> Number of Sequence begins with 1
      BACnetLogRecord listEntry;
}BACnetLogRecordList, *PBACnetLogRecordList;

*)
	nEntrySize	: DWORD; (* 16#80000000 -> next entry *)
	nSequence	: DWORD; (* "reserved"  -> Number OF Sequence begins with 1 *)
	listEntry	: ST_BACnet_LogRecord; (* first entry of record list *)
END_STRUCT
END_TYPE

(* Data type *)
TYPE ST_BACnet_NotificationSinkEventEntry :
STRUCT
	_fillBytes00				: ARRAY[0..7] OF BYTE; (* list header *)
	validFields					: UDINT;	(*	ULONG validFields; *)
	processIdentifier			: UDINT; (*     ULONG processIdentifier; *)
	initiatingDeviceIdentifier	: T_BACnet_ObjectIdentifier; (*  BACnetObjectIdentifier initiatingDeviceIdentifier; *)
	eventObjectIdentifier		: T_BACnet_ObjectIdentifier; (*  BACnetObjectIdentifier eventObjectIdentifier; *)
	timeStamp					: ST_BACnet_TimeStampDateTime;   (* BACnetTimeStamp timeStamp; *)
	notificationClass			: UDINT;  (* ULONG notificationClass;*)
	priority					: UDINT;  (* ULONG priority; *)
	eventType					: E_BACNETEVENTTYPE; (*  BACnetEventType eventType; *)
	_fillBytes01				: WORD; (* fill bytes *)
	messageText					: ARRAY[1..BACnet_STRING_MAXLENGTH] OF BYTE;
	notifyType					: E_BACNETNOTIFYTYPE;  (* BACnetNotifyType notifyType; *)
	_fillBytes02				: WORD; (* fill bytes *)
	ackRequired					: BOOL; (*  BOOL ackRequired; *)
	_fillBytes03				: ARRAY[0..2] OF BYTE; (* fill bytes *)
	fromState					: E_BACNETEVENTSTATE; (*   BACnetEventState fromState; *)
	_fillBytes04				: WORD; (* fill bytes *)
	toState						: E_BACNETEVENTSTATE; (*  BACnetEventState toState; *)
	_fillBytes05				: WORD; (* fill bytes *)
	eventParameterRaw			: ARRAY[0..127] OF BYTE; (* PBACnetNotificationParameters pEventValues; *)
END_STRUCT
END_TYPE

(* Data type *)
TYPE ST_BACnet_NSinkEvent :
STRUCT
	stValidFields	: ST_BACnet_NSinkEventValidFields;
	nProcessID		: UDINT;
	nDeviceID		: UDINT;
	tObjectID		: T_BACnet_ObjectIdentifier;
	stDateTime		: ST_BACnet_DateTime;
	nNC				: UDINT;	(* Notification class object instance *)
	nPriotity		: UDINT;
	eEventType		: E_BACNETEVENTTYPE;
	eNotifyType 	: E_BACNETNOTIFYTYPE;
	eFromState		: E_BACNETEVENTSTATE;
	eToState		: E_BACNETEVENTSTATE;
	sMessage		: T_MaxString;
	bAcknReq		: BOOL; (* Acknowledge required *)
END_STRUCT
END_TYPE

(* Data type *)
TYPE ST_BACnet_NSinkEventValidFields :
STRUCT
      bProcessIdentifier:BOOL; (* Bit0 *)
      bInitiatingDeviceIdentifier:BOOL; (* Bit1 *)
      bEventObjectIdentifier:BOOL; (* Bit2 *)
      bTimeStamp:BOOL; (* Bit3 *)
      bNotificationClass:BOOL; (* Bit4 *)
      bPriority:BOOL; (* Bit5 *)
      bEventType:BOOL; (* Bit6 *)
      bMessageText:BOOL; (* Bit7 *)
      bNotifyType:BOOL; (* Bit8 *)
      bAckRequired:BOOL; (* Bit9 *)
      bFromState:BOOL; (* Bit10 *)
      bToState:BOOL; (* Bit11 *)
      bEventValues:BOOL; (* Bit12 *)
END_STRUCT
END_TYPE

(* Data type *)
TYPE ST_BACnet_ObjectIdentifierList :
STRUCT
	nEntries	: UDINT;
	arrObjList	: ARRAY[0..BACnet_MaxObjIdList] OF T_BACnet_ObjectIdentifier := 16#FFFFFFFF;
END_STRUCT
END_TYPE

(* Data type *)
TYPE ST_BACnet_ObjectTypesSupported:
STRUCT
	SuppAnalogInput : BOOL;
	SuppAnalogOutput : BOOL;
	SuppAnalogValue : BOOL;
	SuppBinaryInput : BOOL;
	SuppBinaryOutput : BOOL;
	SuppBinaryValue : BOOL;
	SuppCalendar : BOOL;
	SuppCommand : BOOL;
	SuppDevice : BOOL;
	SuppEventEnrollment : BOOL;
	SuppFile : BOOL;
	SuppGroup : BOOL;
	SuppLoop : BOOL;
	SuppMultiStateInput : BOOL;
	SuppMultiStateOutput : BOOL;
	SuppNotificationClass : BOOL;
	SuppProgram : BOOL;
	SuppSchedule : BOOL;
	SuppAveraging : BOOL;
	SuppMultiStateValue : BOOL;
	SuppTrendLog : BOOL;
	SuppLifeSafetyPoint : BOOL;
	SuppLifeSafetyZone : BOOL;
END_STRUCT
END_TYPE

(* Data type *)
TYPE ST_BACnet_ProgramHandshakeRequests :
STRUCT
	bLoad	: BOOL;
	bSetup	: BOOL;
	bRun	: BOOL;
	bHalt	: BOOL;
	bUnload	: BOOL;
END_STRUCT
END_TYPE

(* Data type *)
TYPE ST_BACnet_ProgramHandshakeStates :
STRUCT
	bIdle		: BOOL;
	bLoading	: BOOL;
	bRunning	: BOOL;
	bWaiting	: BOOL;
	bHalted		: BOOL;
	bUnloading	: BOOL;
END_STRUCT
END_TYPE

(* Data type *)
TYPE ST_BACnet_RecipientDevice :
STRUCT
	eRecipientChoice: E_BACnetRecipientChoice;
	res				: WORD; (* allignment *)
	tDeviceId		: T_BACnet_ObjectIdentifier := 16#FFFFFFFF;
END_STRUCT
END_TYPE

(* Data type *)
TYPE ST_BACnet_RecipientListDevice :
STRUCT
	nEntries	: INT;
	arrDestList	: ARRAY[0..BACnet_MaxDestinationArray] OF ST_BACnet_RecipientListDeviceEntry;
END_STRUCT
END_TYPE

(* Data type *)
TYPE ST_BACnet_RecipientListDeviceEntry :
STRUCT
	bMonday		: BOOL := TRUE;
	bTuesday	: BOOL := TRUE;
	bWednesday	: BOOL := TRUE;
	bThursday	: BOOL := TRUE;
	bFriday		: BOOL := TRUE;
	bSaturday	: BOOL := TRUE;
	bSunday		: BOOL := TRUE;
	stFromTime	: ST_BACnet_Time :=
		(nHour		:= 0,
		nMinute		:= 0,
		nSecond		:= 0,
		nHundredths := 0);
	stToTime	: ST_BACnet_Time :=
		(nHour		:= 23,
		nMinute		:= 59,
		nSecond		:= 59,
		nHundredths := 99);
	tDeviceId	: T_BACnet_ObjectIdentifier := 16#FFFFFFFF;
	nProcessId	: UDINT;
	bToOffNormal: BOOL := TRUE;
	bToFault	: BOOL := TRUE;
	bToNormal	: BOOL := TRUE;
	bIssueConfirmedNotification	: BOOL;
END_STRUCT
END_TYPE

(* Data type *)
TYPE ST_BACnet_ServerStatistics :
STRUCT
	nOpenRequests: DWORD; (* ULONG *)
	nRequestRetries: DWORD; (* ULONG *)
	nRequestTimeOuts: DWORD; (* ULONG *)
	nPropChanges: DWORD; (* ULONG *)
	nPersistWrites: DWORD; (* ULONG *)
	persistChangeSetId: DWORD; (* ULONG *)
	secpersistNextWrite: DWORD; (* ULONG *)
	persistLastWrite: ST_BACnet_DateTime;
END_STRUCT
END_TYPE

(* Data type *)
TYPE ST_BACnet_ServicesSupported:
STRUCT
	SuppAcknowledgeAlarm : BOOL;
	SuppConfirmedCOVNotification : BOOL;
	SuppConfirmedEventNotification : BOOL;
	SuppGetAlarmSummary : BOOL;
	SuppGetEnrollmentSummary : BOOL;
	SuppSubscribeCOV : BOOL;
	SuppAtomicReadFile : BOOL;
	SuppAtomicWriteFile : BOOL;
	SuppAddListElement : BOOL;
	SuppRemoveListElement : BOOL;
	SuppCreateObject : BOOL;
	SuppDeleteObject : BOOL;
	SuppReadProperty : BOOL;
	SuppReadPropertyConditional : BOOL;
	SuppReadPropertyMultiple : BOOL;
	SuppWriteProperty : BOOL;
	SuppWritePropertyMultiple : BOOL;
	SuppDeviceCommunicationControl : BOOL;
	SuppConfirmedPrivateTransfer : BOOL;
	SuppConfirmedTextMessage : BOOL;
	SuppReinitializeDevice : BOOL;
	SuppVtOpen : BOOL;
	SuppVtClose : BOOL;
	SuppVtData : BOOL;
	SuppAuthenticate : BOOL;
	SuppRequestKey : BOOL;
	SuppIAm : BOOL;
	SuppIHave : BOOL;
	SuppUnconfirmedCOVNotification : BOOL;
	SuppUnconfirmedEventNotification : BOOL;
	SuppUnconfirmedPrivateTransfer : BOOL;
	SuppUnconfirmedTextMessage : BOOL;
	SuppTimeSynchronization : BOOL;
	SuppWhoHas : BOOL;
	SuppWhoIs : BOOL;
	SuppReadRange : BOOL;
	SuppUtcTimeSynchronization : BOOL;
	SuppLifeSafetyOperation : BOOL;
	SuppSubscribeCOVProperty : BOOL;
	SuppGetEventInformation : BOOL;
END_STRUCT
END_TYPE

(* Data type *)
TYPE ST_BACnet_SpecialEventCalendarEntryDate :
STRUCT
(*
	typedef struct _BACnetSpecialEvent
	{
	      BACnetSpecialEventChoice choice;
	      union
	      {
	            BACnetCalendarEntry calendarEntry;
	            BACnetObjectIdentifier calendarReference;
	      };
	      DWORD eventPriority; // DWORD due to alignment
	      DWORD reserved;
	      BACnetTimeValueList listOfTimeValues;
	}BACnetSpecialEvent, *PBACnetSpecialEvent;
*)

	eEventChoice		: E_BACnetSpecialEventChoice;
	nRes1				: WORD; (* ENUM alignment *)
	stCalEntry			: ST_BACnet_CalendarEntryDate;
	nRes2				: DWORD;
	iEventPriority		: DWORD;
	nRes3				: DWORD;
	stListOfTimeValues	: ST_BACnet_TimeValueList;

END_STRUCT
END_TYPE

(* Data type *)
TYPE ST_BACnet_SpecialEventCalendarEntryRange :
STRUCT
(*
	typedef struct _BACnetSpecialEvent
	{
	      BACnetSpecialEventChoice choice;
	      union
	      {
	            BACnetCalendarEntry calendarEntry;
	            BACnetObjectIdentifier calendarReference;
	      };
	      DWORD eventPriority; // DWORD due to alignment
	      DWORD reserved;
	      BACnetTimeValueList listOfTimeValues;
	}BACnetSpecialEvent, *PBACnetSpecialEvent;
*)

	eEventChoice		: E_BACnetSpecialEventChoice;
	nRes1				: WORD; (* ENUM alignment *)
	stCalEntry			: ST_BACnet_CalendarEntryDateRange;
	iEventPriority		: DWORD;
	nRes2				: DWORD;
	stListOfTimeValues	: ST_BACnet_TimeValueList;

END_STRUCT
END_TYPE

(* Data type *)
TYPE ST_BACnet_SpecialEventCalendarEntryWnD :
STRUCT
(*
	typedef struct _BACnetSpecialEvent
	{
	      BACnetSpecialEventChoice choice;
	      union
	      {
	            BACnetCalendarEntry calendarEntry;
	            BACnetObjectIdentifier calendarReference;
	      };
	      DWORD eventPriority; // DWORD due to alignment
	      DWORD reserved;
	      BACnetTimeValueList listOfTimeValues;
	}BACnetSpecialEvent, *PBACnetSpecialEvent;
*)

	eEventChoice		: E_BACnetSpecialEventChoice;
	nRes1				: WORD; (* ENUM alignment *)
	stCalEntry			: ST_BACnet_CalendarEntryWeekNDay;
	nRes2				: DWORD;
	iEventPriority		: DWORD;
	nRes3				: DWORD;
	stListOfTimeValues	: ST_BACnet_TimeValueList;

END_STRUCT
END_TYPE

(* Data type *)
TYPE ST_BACnet_SpecialEventCalendarReference :
STRUCT
(*
	typedef struct _BACnetSpecialEvent
	{
	      BACnetSpecialEventChoice choice;
	      union
	      {
	            BACnetCalendarEntry calendarEntry;
	            BACnetObjectIdentifier calendarReference;
	      };
	      DWORD eventPriority; // DWORD due to alignment
	      DWORD reserved;
	      BACnetTimeValueList listOfTimeValues;
	}BACnetSpecialEvent, *PBACnetSpecialEvent;
*)

	eEventChoice		: E_BACnetSpecialEventChoice;
	nRes1				: WORD; (* ENUM alignment *)
	tCalRef				: T_BACnet_ObjectIdentifier := 16#FFFFFFFF;
	nRes2				: DWORD;
	nRes3				: DWORD;
	iEventPriority		: DWORD;
	nRes4				: DWORD;
	stListOfTimeValues	: ST_BACnet_TimeValueList;

END_STRUCT
END_TYPE

(* Data type *)
TYPE ST_BACnet_SpecialEventListCalEntryDate :
STRUCT
(*
	typedef struct _BACnetSpecialEventList
	{
	      DWORD nEntrySize; // 0x80000000 -> next entry
	      DWORD reserved;
	      BACnetSpecialEvent listEntry;
	}BACnetSpecialEventList, *PBACnetSpecialEventList;
*)
	nEntrySize		: DWORD;
	nRes			: DWORD;
	stListEntry		: ST_BACnet_SpecialEventCalendarEntryDate;
END_STRUCT
END_TYPE

(* Data type *)
TYPE ST_BACnet_SpecialEventListCalEntryRange :
STRUCT
(*
	typedef struct _BACnetSpecialEventList
	{
	      DWORD nEntrySize; // 0x80000000 -> next entry
	      DWORD reserved;
	      BACnetSpecialEvent listEntry;
	}BACnetSpecialEventList, *PBACnetSpecialEventList;
*)
	nEntrySize		: DWORD;
	nRes			: DWORD;
	stListEntry		: ST_BACnet_SpecialEventCalendarEntryRange;
END_STRUCT
END_TYPE

(* Data type *)
TYPE ST_BACnet_SpecialEventListCalEntryWnD :
STRUCT
(*
	typedef struct _BACnetSpecialEventList
	{
	      DWORD nEntrySize; // 0x80000000 -> next entry
	      DWORD reserved;
	      BACnetSpecialEvent listEntry;
	}BACnetSpecialEventList, *PBACnetSpecialEventList;
*)
	nEntrySize		: DWORD;
	nRes			: DWORD;
	stListEntry		: ST_BACnet_SpecialEventCalendarEntryWnD;
END_STRUCT
END_TYPE

(* Data type *)
TYPE ST_BACnet_SpecialEventListCalReference :
STRUCT
(*
	typedef struct _BACnetSpecialEventList
	{
	      DWORD nEntrySize; // 0x80000000 -> next entry
	      DWORD reserved;
	      BACnetSpecialEvent listEntry;
	}BACnetSpecialEventList, *PBACnetSpecialEventList;
*)
	nEntrySize		: DWORD;
	nRes			: DWORD;
	stListEntry		: ST_BACnet_SpecialEventCalendarReference;
END_STRUCT
END_TYPE

(* Data type *)
TYPE ST_BACnet_StatusFlags:
STRUCT
	in_alarm : BOOL;
	fault : BOOL;
	overridden : BOOL;
	out_of_service : BOOL;
END_STRUCT
END_TYPE

(* Data type *)
TYPE ST_BACnet_TcIoEthStatistic :
STRUCT
	dcTimeStamp: ARRAY[0..1] OF DWORD; (* ULONGLONG *)
	sendFrames: DWORD; (* ULONG *)
	recvFrames: DWORD; (* ULONG *)
	sendTimeRTime: DWORD; (* ULONG *)
	recvTimeRTime: DWORD; (* ULONG *)
	sendTimeNdis: DWORD; (* ULONG *)
	recvTimeNdis: DWORD; (* ULONG *)
END_STRUCT
END_TYPE

(* Data type *)
TYPE ST_BACnet_TcIoEthTxRxErrorCount :
STRUCT
	txCnt: DWORD; (* ULONG *)
	rxCnt: DWORD; (* ULONG *)
END_STRUCT
END_TYPE

(* Data type *)
TYPE ST_BACnet_Time :
STRUCT
	nHour		: BYTE := 16#FF; (* hour (0..23), (X'FF') = unspecified *)
	nMinute		: BYTE := 16#FF;	(* minute (0..59), (X'FF') = unspecified *)
	nSecond		: BYTE := 16#FF; (* (0..59), (X'FF') = unspecified *)
	nHundredths	: BYTE := 16#FF;	(* hundredths (0..99), (X'FF') = unspecified *)
END_STRUCT
END_TYPE

(* Data type *)
TYPE ST_BACnet_TimeStampDateTime :
STRUCT
	eType		: E_BACnetTimeStampChoice;
	_fillBytes	: WORD;
	stDateTime	: ST_BACnet_DateTime;
END_STRUCT
END_TYPE

(* Data type *)
TYPE ST_BACnet_TimeValue :
STRUCT
(*
	typedef struct _BACnetTimeValue
	{
	      BACnetTime time;
	      DWORD  reserved;  // 64bit Alignment
	      BACnetValue value;
	}BACnetTimeValue, *PBACnetTimeValue;
*)
	stTime	: ST_BACnet_Time;
	nRes	: DWORD;
	stValue	: ST_BACnet_Value;
END_STRUCT
END_TYPE

(* Data type *)
TYPE ST_BACnet_TimeValueBool :
STRUCT
	bValid		: BOOL;
	stTime		: ST_BACnet_Time;
	eType		: E_BACnetDataTypes;
	bValue		: BOOL;
END_STRUCT
END_TYPE

(* Data type *)
TYPE ST_BACnet_TimeValueList :
STRUCT
(*
	typedef struct _BACnetTimeValueList
	{
	      DWORD nEntrySize; // 0x80000000 -> next entry
	      DWORD reserved;
	      BACnetTimeValue listEntry;
	}BACnetTimeValueList, *PBACnetTimeValueList;
*)
	nEntrySize	: DWORD;
	nRes		: DWORD;
	stListEntry	: ST_BACnet_TimeValue;
END_STRUCT
END_TYPE

(* Data type *)
TYPE ST_BACnet_TimeValueReal :
STRUCT
	bValid		: BOOL;
	stTime		: ST_BACnet_Time;
	eType		: E_BACnetDataTypes;
	rValue		: REAL;
END_STRUCT
END_TYPE

(* Data type *)
TYPE ST_BACnet_UnConfirmedServiceDiag :
STRUCT
	nReqSend: DWORD; (* ULONG *)
	nReqSendFail: DWORD; (* ULONG *)
	nReqRecv: DWORD; (* ULONG *)
	nReqRecvFail: DWORD; (* ULONG *)
END_STRUCT
END_TYPE

(* Data type *)
TYPE ST_BACnet_Value :
STRUCT
(*
	typedef struct _BACnetValue  
	{
	      BACnetValueChoice choice;
	      DWORD                        length;     // Alignment + Datenlänge die folgt
	      union
	      {
	            BOOL                                     boolValue;
	            FLOAT                                    realValue;
	            DOUBLE                                   doubleValue;
	            INT                                      signedValue;
	            UINT                                     unsignedValue;
	            BYTE*                                    pOctedStringValue; 
	            CHAR*                                    pCharStringValue;
	            BACnetObjectIdentifier  objectIdentifierValue;
	            EnumerationValueType         enumerationValue;
	      };
	}BACnetValue, *PBACnetValue;
*)
	eValueChoice	: E_BACnetDataTypes;
	nRes1			: WORD; (* ENUM alignment *)
	cbData			: DWORD;
	nData			: BYTE;

END_STRUCT
END_TYPE

(* Data type *)
TYPE ST_BACnet_WeeklyScheduleBool :
STRUCT
	bReqGet		: BOOL; (* set TRUE if property should reloaded, TRUE --> FALSE = request accepted (reload started) *)
	bReqSet		: BOOL; (* set TRUE for property write request, TRUE --> FALSE = request accepted (storage started) *)
	nGet		: USINT; (* reload counter, count up if property was loaded successful *)
	nSet		: USINT; (* save counter, count up if property was stored successful *)
	bBusy		: BOOL; (* started writing/reading data into/from "arrEntries", don't change data to avoid concurrent access *)
	arrEntries	: ARRAY[0..6] OF ARRAY[0..BACnet_MaxDayEntry] OF ST_BACnet_TimeValueBool;
END_STRUCT
END_TYPE

(* Data type *)
TYPE ST_BACnet_WeeklyScheduleReal :
STRUCT
	bReqGet		: BOOL; (* set TRUE if property should reloaded, TRUE --> FALSE = request accepted (reload started) *)
	bReqSet		: BOOL; (* set TRUE for property write request, TRUE --> FALSE = request accepted (storage started) *)
	nGet		: USINT; (* reload counter, count up if property was loaded successful *)
	nSet		: USINT; (* save counter, count up if property was stored successful *)
	bBusy		: BOOL; (* started writing/reading data into/from "arrEntries", don't change data to avoid concurrent access *)
	arrEntries	: ARRAY[0..6] OF ARRAY[0..BACnet_MaxDayEntry] OF ST_BACnet_TimeValueReal;
END_STRUCT
END_TYPE

(* Data type *)
TYPE T_BACnet_CalendarEntryTypeFilter : ARRAY[0..4] OF E_BACnetCalendarEntryType; END_TYPE

(* Data type *)
TYPE T_BACnet_DestinationDeviceArray : ARRAY[0..BACnet_MaxDestinationArray] OF ST_BACnet_DestinationDevice; END_TYPE

(* Data type *)
TYPE T_BACnet_ObjectIdentifier : DWORD; END_TYPE

(* POU _F_BACnet_AlignedSize, ST *)
FUNCTION _F_BACnet_AlignedSize : DWORD
VAR_INPUT
	n	: DWORD;
END_VAR
VAR
END_VAR
_F_BACnet_AlignedSize := (4*(((n)+3)/4));
END_FUNCTION

(* POU _F_BACnet_BitFieldBit, ST *)
FUNCTION _F_BACnet_BitFieldBit : WORD
VAR_INPUT
	Bit	:	WORD;
END_VAR
VAR
END_VAR
_F_BACnet_BitFieldBit := (Bit/8) * 8 + (bit MOD 8);
END_FUNCTION

(* POU _F_BACnet_ChangeBitFieldBit, ST *)
FUNCTION _F_BACnet_ChangeBitFieldBit : DWORD
VAR_INPUT
	ptrData		: POINTER TO DWORD;
	Bit			: WORD;
	Value		: BOOL;
END_VAR
VAR
END_VAR
IF (NOT Value) THEN
	ptrData^ := ptrData^ AND NOT (SHR(DWORD#16#00008000,_F_BACnet_BitFieldBit(Bit)));
ELSE
	ptrData^ := ptrData^ OR (SHR(DWORD#16#00008000,_F_BACnet_BitFieldBit(Bit)));
END_IF
_F_BACnet_ChangeBitFieldBit := ptrData^;
END_FUNCTION

(* POU _F_BACnet_ChrStrExtLen, ST *)
FUNCTION _F_BACnet_ChrStrExtLen : UDINT
VAR_IN_OUT
	stCharStringExt	: ST_BACnet_CharacterStringExt;
END_VAR
VAR
	pByte	: POINTER TO BYTE;
	nLen	: UDINT;
END_VAR
pByte := ADR(stCharStringExt);
nLen := SIZEOF(stCharStringExt);
(* check the string type *)
IF (nLen > 4 AND stCharStringExt.cookie = 0) THEN
	(* character string ext. *)
	IF (stCharStringExt.strLen <= SIZEOF(stCharStringExt.stringData)) THEN
		(* plausible string length given *)
		_F_BACnet_ChrStrExtLen := stCharStringExt.strLen;
		RETURN;
	END_IF
	(* use sizeof, because string length isn't plausible *)
	nLen := SIZEOF(stCharStringExt.stringData);
	(* re-adjust pointer *)
	pByte := ADR(stCharStringExt.stringData);
END_IF
(* scan zero termination *)
_F_BACnet_ChrStrExtLen := 0;
WHILE ((pByte^ <> 0) AND (_F_BACnet_ChrStrExtLen < nLen)) DO
	pByte := pByte + 1;
	_F_BACnet_ChrStrExtLen := _F_BACnet_ChrStrExtLen + 1;
END_WHILE
END_FUNCTION

(* POU _F_BACnet_DecodeUCS2, ST *)
FUNCTION _F_BACnet_DecodeUCS2 : UDINT (* result is the new character length of the string *)
VAR_INPUT
	pString		: POINTER TO WORD; (* pointer to UCS2 string beginning *)
	cbString	: UDINT; (* byte size of string (use SIZEOF - don't use LEN) *)
END_VAR
VAR
	i		: UDINT;
	pResult	: POINTER TO BYTE;
	pBy		: POINTER TO WORD;
END_VAR
pResult	:= pString;
pBy		:= pString;
FOR i := 0 TO cbString-1 DO
	pResult^ := _F_BACnet_UCS2ToWin1252(pBy, TRUE);
	pBy := pBy + 2;
	(* end-of-string by character *)
	IF (pResult^ = 16#00) THEN
		EXIT;
	END_IF
	(* next character *)
	pResult := pResult + 1;
	(* end-of-string by length *)
	IF (pBy >= (pString + cbString)) THEN
		EXIT;
	END_IF
END_FOR
pResult^ := 16#00;
_F_BACnet_DecodeUCS2 := pResult - pString;
END_FUNCTION

(* POU _F_BACnet_UCS2ToWin1252, ST *)
FUNCTION _F_BACnet_UCS2ToWin1252 : BYTE
VAR_INPUT
	pUCS2 :	POINTER TO WORD;
	bBE	: BOOL; (* byte-order big endian = TRUE *)
END_VAR
VAR
	pArr : POINTER TO ARRAY[0..1] OF BYTE;
	wUCS2: WORD;
END_VAR
VAR CONSTANT
	cRepl	: BYTE := 16#5F;
END_VAR
(*
	Windows-Codepages
874		Thai
932		Japanisch
936		Vereinfachtes Chinesisch
949		Koreanisch
950		Traditionelles Chinesisch
1250	Mitteleuropäisch
1251	Kyrillisch
1252	Westeuropäisch
1253	Griechisch
1254	Türkisch
1255	Hebräisch
1256	Arabisch
1257	Baltisch
1258	Vietnamesisch
*)
pArr := pUCS2;
IF bBE THEN
	wUCS2 := (pArr^[0] * 16#0100) + pArr^[1];
ELSE
	wUCS2 := pUCS2^;
END_IF
CASE wUCS2 OF
	16#178: 	_F_BACnet_UCS2ToWin1252 := 16#9F;
	16#153: 	_F_BACnet_UCS2ToWin1252 := 16#9C;
	16#152: 	_F_BACnet_UCS2ToWin1252 := 16#8C;
	16#17E: 	_F_BACnet_UCS2ToWin1252 := 16#9E;
	16#17D: 	_F_BACnet_UCS2ToWin1252 := 16#8E;
	16#161: 	_F_BACnet_UCS2ToWin1252 := 16#9A;
	16#160: 	_F_BACnet_UCS2ToWin1252 := 16#8A;
	16#20AC: 	_F_BACnet_UCS2ToWin1252 := 16#80;
	ELSE
		IF wUCS2 <= 16#FF THEN
			_F_BACnet_UCS2ToWin1252 := WORD_TO_BYTE(wUCS2);
		ELSE
			_F_BACnet_UCS2ToWin1252 := cRepl;
		END_IF
END_CASE
END_FUNCTION

(* POU _F_BACnet_DecodeUCS4, ST *)
FUNCTION _F_BACnet_DecodeUCS4 : UDINT (* result is the new character length of the string *)
VAR_INPUT
	pString		: POINTER TO DWORD; (* pointer to UCS4 string beginning *)
	cbString	: UDINT; (* byte size of string (use SIZEOF - don't use LEN) *)
END_VAR
VAR
	i		: UDINT;
	pResult	: POINTER TO BYTE;
	pBy		: POINTER TO WORD;
END_VAR
pResult	:= pString;
pBy		:= pString;
FOR i := 0 TO cbString-1 DO
	(* byte order big endian *)
	pResult^ := _F_BACnet_UCS2ToWin1252(pBy+2, TRUE);
	pBy := pBy + 4;
	(* end-of-string by character *)
	IF (pResult^ = 16#00) THEN
		EXIT;
	END_IF
	(* next character *)
	pResult := pResult + 1;
	(* end-of-string by length *)
	IF (pBy >= (pString + cbString)) THEN
		EXIT;
	END_IF
END_FOR
pResult^ := 16#00;
_F_BACnet_DecodeUCS4 := pResult - pString;
END_FUNCTION

(* POU _F_BACnet_DecodeUTF8, ST *)
FUNCTION _F_BACnet_DecodeUTF8 : UDINT (* result is the new character length of the string *)
VAR_INPUT
	pString		: POINTER TO BYTE; (* pointer to UTF-8 string beginning *)
	cbString	: UDINT; (* byte size of string (use SIZEOF - don't use LEN) *)
END_VAR
VAR
	i			: UDINT;
	pResult		: POINTER TO BYTE;
	pBy			: POINTER TO BYTE;
	pByArr		: POINTER TO ARRAY[0..3] OF BYTE;
END_VAR
pResult	:= pString;
pBy		:= pString;
FOR i := 0 TO cbString-1 DO
	pByArr := pBy;
	IF (pByArr^[0] AND 16#F0) = 16#C0 THEN
		IF (pByArr^[1] AND 16#80) = 16#80 THEN
			pResult^ := _F_BACnet_Utf8ToWin1252(pByArr, 2);
			pBy := pBy + 2;
		END_IF
	ELSIF (pByArr^[0] AND 16#F0) = 16#E0 THEN
		IF (pByArr^[1] AND 16#80) = 16#80 THEN
			IF (pByArr^[2] AND 16#80) = 16#80 THEN
				pResult^ := _F_BACnet_Utf8ToWin1252(pByArr, 3);
				pBy := pBy + 3;
			END_IF
		END_IF
	ELSIF (pByArr^[0] AND 16#F0) = 16#F0 THEN
		IF (pByArr^[1] AND 16#80) = 16#80 THEN
			IF (pByArr^[2] AND 16#80) = 16#80 THEN
				IF (pByArr^[3] AND 16#80) = 16#80 THEN
					pResult^ := _F_BACnet_Utf8ToWin1252(pByArr, 4);
					pBy := pBy + 4;
				END_IF
			END_IF
		END_IF
	ELSE
		(* ASCII character *)
		pResult^ := pBy^;
		pBy := pBy + 1;
	END_IF
	(* end-of-string by character *)
	IF (pResult^ = 16#00) THEN
		EXIT;
	END_IF
	(* next character *)
	pResult := pResult + 1;
	(* end-of-string by length *)
	IF (pBy >= (pString + cbString)) THEN
		EXIT;
	END_IF
END_FOR
pResult^ := 16#00;
_F_BACnet_DecodeUTF8 := pResult - pString;
END_FUNCTION

(* POU _F_BACnet_Utf8ToWin1252, ST *)
FUNCTION _F_BACnet_Utf8ToWin1252 : BYTE
VAR_INPUT
	pUtf8	: POINTER TO BYTE;
	cbUtf8	: UDINT; (* byte size of UTF8 character (1...6) *)
END_VAR
VAR
	pArr		: POINTER TO ARRAY[0..5] OF BYTE;
	pWord		: POINTER TO ARRAY[0..1] OF BYTE;
	wUCS2		: WORD;
END_VAR
VAR CONSTANT
	cRepl	: BYTE := 16#5F;
END_VAR
(*
	Windows-Codepages
874		Thai
932		Japanisch
936		Vereinfachtes Chinesisch
949		Koreanisch
950		Traditionelles Chinesisch
1250	Mitteleuropäisch
1251	Kyrillisch
1252	Westeuropäisch
1253	Griechisch
1254	Türkisch
1255	Hebräisch
1256	Arabisch
1257	Baltisch
1258	Vietnamesisch
*)
(* first step - convert to UCS2 *)
pArr := pUtf8;
IF (pArr^[0] <= 16#7F) THEN
	(* basic latin *)
	_F_BACnet_Utf8ToWin1252 := pArr^[0];
	RETURN;
ELSIF (cbUtf8 >= 2) THEN
	pWord := ADR(wUCS2);
	IF (pArr^[0] = 16#C2) THEN
		(* latin-1 supplement *)
		wUCS2 := pArr^[1];
	ELSIF (pArr^[0] = 16#C3) AND (pArr^[1] <= 16#BF) THEN
		(* latin-1 supplement *)
		wUCS2 := pArr^[1] + 16#40;
	ELSIF (pArr^[0] = 16#C4) AND (pArr^[1] >= 16#80) THEN
		(* latin extended-A *)
		pWord^[1] := 16#01;
		pWord^[0] := pArr^[1] - 16#80;
	ELSIF (pArr^[0] = 16#C5) AND (pArr^[1] >= 16#80) THEN
		(* latin extended-A *)
		pWord^[1] := 16#01;
		pWord^[0] := pArr^[1] - 16#40;
	ELSIF (pArr^[0] = 16#C6) AND (pArr^[1] >= 16#80) THEN
		(* latin extended-B *)
		pWord^[1] := 16#01;
		pWord^[0] := pArr^[1];
	ELSIF (pArr^[0] = 16#C7) AND (pArr^[1] <= 16#BF) THEN
		(* latin extended-B *)
		pWord^[1] := 16#01;
		pWord^[0] := pArr^[1] + 16#40;
	ELSIF (cbUtf8 >= 3) THEN
		IF (pArr^[0] = 16#E2) AND (pArr^[1] = 16#82) THEN
			(* currency symbols *)
			pWord^[1] := 16#20;
			pWord^[0] := pArr^[2];
		ELSE
			(* unsupported *)
			_F_BACnet_Utf8ToWin1252 := cRepl;
			RETURN;
		END_IF
	ELSE
		(* unsupported *)
		_F_BACnet_Utf8ToWin1252 := cRepl;
		RETURN;
	END_IF
	(* convert UCS2 to Windows-1252 *)
	_F_BACnet_Utf8ToWin1252 := _F_BACnet_UCS2ToWin1252(pWord, FALSE);
	RETURN;
END_IF
(* unsupported *)
_F_BACnet_Utf8ToWin1252 := cRepl;
END_FUNCTION

(* POU _F_BACnet_EncodeUTF8, ST *)
FUNCTION _F_BACnet_EncodeUTF8 : UDINT (* actually byte length of the result utf-8 string (maybe longer than cbResult; means overflow) *)
VAR_INPUT
	pString		: POINTER TO BYTE; (* pointer to Win1252 string beginning *)
	cbString	: UDINT; (* byte size of string (use SIZEOF - don't use LEN) *)
	pResult		: POINTER TO BYTE; (* pointer to result UTF-8 data area *)
	cbResult	: UDINT; (* byte size of result (use SIZEOF - don't use LEN) *)
END_VAR
VAR_IN_OUT
	nResultLen	: UDINT; (* final resulting string length (<= cbResult) *)
END_VAR
VAR
	pBy			: POINTER TO BYTE;
	pByArr		: POINTER TO ARRAY[0..3] OF BYTE;
	nCoded		: UINT;
	bOverflow	: BOOL;
END_VAR
pBy			:= pString;
pByArr		:= pResult;
bOverflow	:= FALSE;
_F_BACnet_EncodeUTF8 := 0;
nResultLen	:= 0;
(* loop over pString *)
WHILE pBy < (pString + cbString) DO
	IF (pBy^ = 0) THEN EXIT; END_IF
	IF bOverflow OR (_F_BACnet_EncodeUTF8 + 3 > cbResult) THEN
		nCoded := _F_BACnet_Win1252ToUtf8(nW1252:=pBy^, pUtf8:=pByArr, bEval:=TRUE);
		IF (NOT bOverflow) AND (_F_BACnet_EncodeUTF8 + nCoded <= cbResult) THEN
			nCoded := _F_BACnet_Win1252ToUtf8(nW1252:=pBy^, pUtf8:=pByArr, bEval:=FALSE);
		ELSE
			bOverflow := TRUE;
		END_IF
	ELSE
		nCoded := _F_BACnet_Win1252ToUtf8(nW1252:=pBy^, pUtf8:=pByArr, bEval:=FALSE);
	END_IF
	IF (NOT bOverflow) THEN
		pByArr := pByArr + UINT_TO_UDINT(nCoded);
		nResultLen := _F_BACnet_EncodeUTF8 + nCoded;
	END_IF
	_F_BACnet_EncodeUTF8 := _F_BACnet_EncodeUTF8 + nCoded;
	pBy := pBy + 1;
END_WHILE
(* add zero termination if needed *)
IF (nResultLen < cbResult) THEN
	pByArr^[0] := 16#00;
END_IF
END_FUNCTION

(* POU _F_BACnet_Win1252ToUtf8, ST *)
FUNCTION _F_BACnet_Win1252ToUtf8 : UINT(0..3)
VAR_INPUT
	nW1252	: BYTE; (* Win1252 character *)
	pUtf8	: POINTER TO ARRAY[0..2] OF BYTE; (* pointer to target character buffer (utf-8) *)
	bEval	: BOOL; (* TRUE = only evaluate expected coding size (0..3 byte) - but don't write data *)
END_VAR
VAR
	pWord	: POINTER TO ARRAY[0..1] OF BYTE;
	wUCS2	: WORD;
END_VAR
VAR CONSTANT
	cRepl	: BYTE := 16#5F;
END_VAR
(*
	Windows-Codepages
874		Thai
932		Japanisch
936		Vereinfachtes Chinesisch
949		Koreanisch
950		Traditionelles Chinesisch
1250	Mitteleuropäisch
1251	Kyrillisch
1252	Westeuropäisch
1253	Griechisch
1254	Türkisch
1255	Hebräisch
1256	Arabisch
1257	Baltisch
1258	Vietnamesisch
*)
(* check pointer *)
IF (pUtf8 = 0) THEN
	(* null pointer *)
	_F_BACnet_Win1252ToUtf8 := 0;
ELSIF (nW1252 <= 16#7F) THEN
	(* basic latin - 1 byte *)
	IF (NOT bEval) THEN
		pUtf8^[0] := nW1252;
	END_IF
	_F_BACnet_Win1252ToUtf8 := 1;
ELSE
	(* convert to UCS-2 first *)
	wUCS2 := _F_BACnet_Win1252ToUCS2(nW1252:=nW1252, bBE:=FALSE);
	pWord := ADR(wUCS2);
	(* convert used ranges *)
	IF (wUCS2 >= 16#80 AND wUCS2 <= 16#BF) THEN
		(* latin-1 supplement *)
		IF (NOT bEval) THEN
			pUtf8^[0] := 16#C2;
			pUtf8^[1] := pWord^[0];
		END_IF
		_F_BACnet_Win1252ToUtf8 := 2;
	ELSIF (wUCS2 >= 16#C0 AND wUCS2 <= 16#FF) THEN
		(* latin-1 supplement *)
		IF (NOT bEval) THEN
			pUtf8^[0] := 16#C3;
			pUtf8^[1] := pWord^[0] - 16#40;
		END_IF
		_F_BACnet_Win1252ToUtf8 := 2;
	ELSIF (wUCS2 >= 16#140 AND wUCS2 <= 16#17F) THEN
		(* latin extended A *)
		IF (NOT bEval) THEN
			pUtf8^[0] := 16#C5;
			pUtf8^[1] := pWord^[0] + 16#40;
		END_IF
		_F_BACnet_Win1252ToUtf8 := 2;
	ELSIF (wUCS2 >= 16#20A0 AND wUCS2 <= 16#20BF) THEN
		(* currency symbols *)
		IF (NOT bEval) THEN
			pUtf8^[0] := 16#E2;
			pUtf8^[1] := 16#82;
			pUtf8^[2] := pWord^[0];
		END_IF
		_F_BACnet_Win1252ToUtf8 := 3;
	ELSE
		(* unsupported *)
		IF (NOT bEval) THEN
			pUtf8^[0] := cRepl;
		END_IF
		_F_BACnet_Win1252ToUtf8 := 1;
	END_IF
END_IF
END_FUNCTION

(* POU _F_BACnet_Win1252ToUCS2, ST *)
FUNCTION _F_BACnet_Win1252ToUCS2 : WORD
VAR_INPUT
	nW1252 : BYTE;
	bBE	: BOOL; (* byte-order big endian = TRUE *)
END_VAR
VAR
	pArr : POINTER TO ARRAY[0..1] OF BYTE;
	nBuf : BYTE;
	wUCS2: WORD;
END_VAR
(*
	Windows-Codepages
874		Thai
932		Japanisch
936		Vereinfachtes Chinesisch
949		Koreanisch
950		Traditionelles Chinesisch
1250	Mitteleuropäisch
1251	Kyrillisch
1252	Westeuropäisch
1253	Griechisch
1254	Türkisch
1255	Hebräisch
1256	Arabisch
1257	Baltisch
1258	Vietnamesisch
*)
CASE nW1252 OF
	16#9F: wUCS2 := 16#178;
	16#9C: wUCS2 := 16#153;
	16#8C: wUCS2 := 16#152;
	16#9E: wUCS2 := 16#17E;
	16#8E: wUCS2 := 16#17D;
	16#9A: wUCS2 := 16#161;
	16#8A: wUCS2 := 16#160;
	16#80: wUCS2 := 16#20AC;
	ELSE
	wUCS2 := nW1252;
END_CASE
IF bBE THEN
	pArr := ADR(wUCS2);
	nBuf := pArr^[0];
	pArr^[0] := pArr^[1];
	pArr^[1] := nBuf;
END_IF
_F_BACnet_Win1252ToUCS2 := wUCS2;
END_FUNCTION

(* POU _F_BACnet_IsBitFieldBitSet, ST *)
FUNCTION _F_BACnet_IsBitFieldBitSet : BOOL
VAR_INPUT
	data	:	DWORD;
	Bit		:	WORD;
END_VAR
VAR
END_VAR
_F_BACnet_IsBitFieldBitSet:= (data AND (SHR(DWORD#16#00008000,_F_BACnet_BitFieldBit(Bit)))) > 0;
END_FUNCTION

(* POU _F_BACnet_SetBitFieldBit, ST *)
FUNCTION _F_BACnet_SetBitFieldBit : DWORD
VAR_INPUT
	ptrData		:	POINTER TO DWORD;
	Bit			:	WORD;
END_VAR
VAR
END_VAR
ptrData^ := ptrData^ OR (SHR(DWORD#16#00008000, _F_BACnet_BitFieldBit(Bit)));
_F_BACnet_SetBitFieldBit := ptrData^;
END_FUNCTION

(* POU _F_BACnet_SysTimeDiff, ST *)
FUNCTION _F_BACnet_SysTimeDiff : REAL
VAR_INPUT
	In1, In2 : T_LARGE_INTEGER;
END_VAR
_F_BACnet_SysTimeDiff := LREAL_TO_REAL(INT64_TO_LREAL(Int64Sub64(In1, In2)) / 10000000.0); (* [s] *)
END_FUNCTION

(* POU _F_BACnet_UnSetBitFieldBit, ST *)
FUNCTION _F_BACnet_UnSetBitFieldBit : DWORD
VAR_INPUT
	ptrData		:	POINTER TO DWORD;
	Bit			:	WORD;
END_VAR
VAR
END_VAR
ptrData^ := ptrData^ AND NOT (SHR(DWORD#16#00008000,_F_BACnet_BitFieldBit(Bit)));
_F_BACnet_UnSetBitFieldBit := ptrData^;
END_FUNCTION

